LIN {X 0,Y 145.959,Z 433.252,A -85,B 0,C 180,E1 -25512.385,E2 -25512.385} C_VEL
LIN {X 0,Y 151.822,Z 425.901,A -85,B 0,C 180,E1 -25515.592,E2 -25515.592} C_VEL
LIN {X 0,Y 158.562,Z 416.452,A -85,B 0,C 180,E1 -25518.895,E2 -25518.895} C_VEL
LIN {X 0,Y 165.615,Z 405.723,A -85,B 0,C 180,E1 -25521.727,E2 -25521.727} C_VEL
LIN {X 0,Y 172.327,Z 394.008,A -85,B 0,C 180,E1 -25524.151,E2 -25524.151} C_VEL
LIN {X 0,Y 178.873,Z 380.825,A -85,B 0,C 180,E1 -25526.236,E2 -25526.236} C_VEL
LIN {X 0,Y 184.461,Z 367.074,A -85,B 0,C 180,E1 -25527.966,E2 -25527.966} C_VEL
LIN {X 0,Y 189.113,Z 353.283,A -85,B 0,C 180,E1 -25529.249,E2 -25529.249} C_VEL
LIN {X 0,Y 193.148,Z 337.834,A -85,B 0,C 180,E1 -25530.312,E2 -25530.312} C_VEL
LIN {X 0,Y 196.132,Z 321.975,A -85,B 0,C 180,E1 -25531.033,E2 -25531.033} C_VEL
LIN {X 0,Y 198.364,Z 301.16,A -85,B 0,C 180,E1 -25531.651,E2 -25531.651} C_VEL
LIN {X 0,Y 201.461,Z 266.459,A -85,B 0,C 180,E1 -25532.587,E2 -25532.587} C_VEL
LIN {X 0,Y 197.2,Z 257.514,A -85,B 0,C 180,E1 -25535.874,E2 -25535.874} C_VEL
LIN {X 0,Y 193.615,Z 250.815,A -85,B 0,C 180,E1 -25539.064,E2 -25539.064} C_VEL
LIN {X 0,Y 191.118,Z 246.438,A -85,B 0,C 180,E1 -25541.647,E2 -25541.647} C_VEL
LIN {X 0,Y 189.084,Z 243.025,A -85,B 0,C 180,E1 -25544.09,E2 -25544.09} C_VEL
LIN {X 0,Y 187.689,Z 240.639,A -85,B 0,C 180,E1 -25546.051,E2 -25546.051} C_VEL
LIN {X 0,Y 185.533,Z 236.807,A -85,B 0,C 180,E1 -25549.91,E2 -25549.91} C_VEL
LIN {X 0,Y 183.726,Z 233.495,A -85,B 0,C 180,E1 -25555.359,E2 -25555.359} C_VEL
LIN {X 0,Y 183.496,Z 232.327,A -85,B 0,C 180,E1 -25557.256,E2 -25557.256} C_VEL
LIN {X 0,Y 183.478,Z 232.249,A -85,B 0,C 180,E1 -25562.195,E2 -25562.195} C_VEL
LIN {X 0,Y 183.641,Z 233.069,A -85,B 0,C 180,E1 -25563.703,E2 -25563.703} C_VEL
LIN {X 0,Y 185.447,Z 236.708,A -85,B 0,C 180,E1 -25569.566,E2 -25569.566} C_VEL
LIN {X 0,Y 186.036,Z 237.651,A -85,B 0,C 180,E1 -25570.761,E2 -25570.761} C_VEL
LIN {X 0,Y 188.522,Z 241.906,A -85,B 0,C 180,E1 -25574.781,E2 -25574.781} C_VEL
LIN {X 0,Y 190.791,Z 245.771,A -85,B 0,C 180,E1 -25577.622,E2 -25577.622} C_VEL
LIN {X 0,Y 194.145,Z 251.69,A -85,B 0,C 180,E1 -25581.084,E2 -25581.084} C_VEL
LIN {X 0,Y 196.253,Z 256.423,A -85,B 0,C 180,E1 -25583.047,E2 -25583.047} C_VEL
LIN {X 0,Y 199.614,Z 265.237,A -85,B 0,C 180,E1 -25585.917,E2 -25585.917} C_VEL
LIN {X 0,Y 201.239,Z 269.895,A -85,B 0,C 180,E1 -25587.203,E2 -25587.203} C_VEL
LIN {X 0,Y 196.188,Z 324.073,A -85,B 0,C 180,E1 -25588.669,E2 -25588.669} C_VEL
LIN {X 0,Y 193.418,Z 339.856,A -85,B 0,C 180,E1 -25589.301,E2 -25589.301} C_VEL
LIN {X 0,Y 189.561,Z 355.077,A -85,B 0,C 180,E1 -25590.195,E2 -25590.195} C_VEL
LIN {X 0,Y 185.028,Z 368.798,A -85,B 0,C 180,E1 -25591.281,E2 -25591.281} C_VEL
LIN {X 0,Y 179.611,Z 382.244,A -85,B 0,C 180,E1 -25592.725,E2 -25592.725} C_VEL
LIN {X 0,Y 173.675,Z 394.769,A -85,B 0,C 180,E1 -25594.508,E2 -25594.508} C_VEL
LIN {X 0,Y 166.779,Z 407.28,A -85,B 0,C 180,E1 -25596.807,E2 -25596.807} C_VEL
LIN {X 0,Y 159.476,Z 418.758,A -85,B 0,C 180,E1 -25599.537,E2 -25599.537} C_VEL
LIN {X 0,Y 152.629,Z 428.424,A -85,B 0,C 180,E1 -25602.545,E2 -25602.545} C_VEL
LIN {X 0,Y 146.12,Z 436.937,A -85,B 0,C 180,E1 -25605.972,E2 -25605.972} C_VEL
LIN {X 0,Y 139.136,Z 445.526,A -85,B 0,C 180,E1 -25610.542,E2 -25610.542} C_VEL
LIN {X 0,Y 132.201,Z 453.257,A -85,B 0,C 180,E1 -25616.069,E2 -25616.069} C_VEL
LIN {X 0,Y 127.36,Z 458.667,A -85,B 0,C 180,E1 -25621.39,E2 -25621.39} C_VEL
LIN {X 0,Y 125.001,Z 460.669,A -85,B 0,C 180,E1 -25623.685,E2 -25623.685} C_VEL
LIN {X 0,Y 119.759,Z 463.482,A -85,B 0,C 180,E1 -25627.41,E2 -25627.41} C_VEL
LIN {X 0,Y 115.772,Z 465.343,A -85,B 0,C 180,E1 -25630.644,E2 -25630.644} C_VEL
LIN {X 0,Y 113.77,Z 466.536,A -85,B 0,C 180,E1 -25633.365,E2 -25633.365} C_VEL
LIN {X 0,Y 113.419,Z 466.836,A -85,B 0,C 180,E1 -25634.326,E2 -25634.326} C_VEL
LIN {X 0,Y 112.458,Z 468.336,A -85,B 0,C 180,E1 -25639.194,E2 -25639.194} C_VEL
LIN {X 0,Y 112.095,Z 469.523,A -85,B 0,C 180,E1 -25646.405,E2 -25646.405} C_VEL
LIN {X 0,Y 112.248,Z 469.683,A -85,B 0,C 180,E1 -25650,E2 -25650} C_VEL
LIN {X 0,Y 112.127,Z 469.052,A -85,B 0,C 180,E1 -25657.201,E2 -25657.201} C_VEL
LIN {X 0,Y 113.102,Z 467.265,A -85,B 0,C 180,E1 -25664.392,E2 -25664.392} C_VEL
LIN {X 0,Y 115.542,Z 464.307,A -85,B 0,C 180,E1 -25671.405,E2 -25671.405} C_VEL
LIN {X 0,Y 119.379,Z 460.108,A -85,B 0,C 180,E1 -25678.097,E2 -25678.097} C_VEL
LIN {X 0,Y 124.74,Z 454.565,A -85,B 0,C 180,E1 -25684.292,E2 -25684.292} C_VEL
LIN {X 0,Y 131.461,Z 447.53,A -85,B 0,C 180,E1 -25689.906,E2 -25689.906} C_VEL
LIN {X 0,Y 138.147,Z 439.961,A -85,B 0,C 180,E1 -25694.428,E2 -25694.428} C_VEL
LIN {X 0,Y 145.577,Z 430.948,A -85,B 0,C 180,E1 -25698.443,E2 -25698.443} C_VEL
LIN {X 0,Y 153.784,Z 420.066,A -85,B 0,C 180,E1 -25702.03,E2 -25702.03} C_VEL
LIN {X 0,Y 161.304,Z 408.87,A -85,B 0,C 180,E1 -25704.78,E2 -25704.78} C_VEL
LIN {X 0,Y 168.57,Z 396.421,A -85,B 0,C 180,E1 -25707.123,E2 -25707.123} C_VEL
LIN {X 0,Y 175.185,Z 383.102,A -85,B 0,C 180,E1 -25709.039,E2 -25709.039} C_VEL
LIN {X 0,Y 180.735,Z 369.84,A -85,B 0,C 180,E1 -25710.467,E2 -25710.467} C_VEL
LIN {X 0,Y 185.714,Z 355.323,A -85,B 0,C 180,E1 -25711.625,E2 -25711.625} C_VEL
LIN {X 0,Y 189.658,Z 340.259,A -85,B 0,C 180,E1 -25712.503,E2 -25712.503} C_VEL
LIN {X 0,Y 192.438,Z 324.99,A -85,B 0,C 180,E1 -25713.123,E2 -25713.123} C_VEL
LIN {X 0,Y 196.109,Z 288.872,A -85,B 0,C 180,E1 -25714.062,E2 -25714.062} C_VEL
LIN {X 0,Y 197.581,Z 272.685,A -85,B 0,C 180,E1 -25714.504,E2 -25714.504} C_VEL
LIN {X 0,Y 194.287,Z 263.272,A -85,B 0,C 180,E1 -25717.468,E2 -25717.468} C_VEL
LIN {X 0,Y 192.199,Z 258.069,A -85,B 0,C 180,E1 -25719.533,E2 -25719.533} C_VEL
LIN {X 0,Y 189.081,Z 252.283,A -85,B 0,C 180,E1 -25722.91,E2 -25722.91} C_VEL
LIN {X 0,Y 186.331,Z 247.346,A -85,B 0,C 180,E1 -25726.643,E2 -25726.643} C_VEL
LIN {X 0,Y 184.285,Z 243.616,A -85,B 0,C 180,E1 -25730.396,E2 -25730.396} C_VEL
LIN {X 0,Y 182.602,Z 240.468,A -85,B 0,C 180,E1 -25735.447,E2 -25735.447} C_VEL
LIN {X 0,Y 182.361,Z 239.282,A -85,B 0,C 180,E1 -25737.239,E2 -25737.239} C_VEL
LIN {X 0,Y 182.233,Z 239.216,A -85,B 0,C 180,E1 -25742.21,E2 -25742.21} C_VEL
LIN {X 0,Y 182.442,Z 239.623,A -85,B 0,C 180,E1 -25743.866,E2 -25743.866} C_VEL
LIN {X 0,Y 183.716,Z 242.998,A -85,B 0,C 180,E1 -25748.802,E2 -25748.802} C_VEL
LIN {X 0,Y 184.522,Z 244.089,A -85,B 0,C 180,E1 -25750.562,E2 -25750.562} C_VEL
LIN {X 0,Y 186.922,Z 248.505,A -85,B 0,C 180,E1 -25754.702,E2 -25754.702} C_VEL
LIN {X 0,Y 189.301,Z 252.766,A -85,B 0,C 180,E1 -25757.8,E2 -25757.8} C_VEL
LIN {X 0,Y 192.242,Z 258.192,A -85,B 0,C 180,E1 -25760.952,E2 -25760.952} C_VEL
LIN {X 0,Y 195.843,Z 265.523,A -85,B 0,C 180,E1 -25764.233,E2 -25764.233} C_VEL
LIN {X 0,Y 197.761,Z 269.785,A -85,B 0,C 180,E1 -25765.805,E2 -25765.805} C_VEL
LIN {X 0,Y 192.923,Z 319.693,A -85,B 0,C 180,E1 -25767.155,E2 -25767.155} C_VEL
LIN {X 0,Y 190.163,Z 335.085,A -85,B 0,C 180,E1 -25767.788,E2 -25767.788} C_VEL
LIN {X 0,Y 186.696,Z 349.013,A -85,B 0,C 180,E1 -25768.648,E2 -25768.648} C_VEL
LIN {X 0,Y 182.267,Z 362.803,A -85,B 0,C 180,E1 -25769.822,E2 -25769.822} C_VEL
LIN {X 0,Y 176.796,Z 376.715,A -85,B 0,C 180,E1 -25771.409,E2 -25771.409} C_VEL
LIN {X 0,Y 170.343,Z 390.076,A -85,B 0,C 180,E1 -25773.335,E2 -25773.335} C_VEL
LIN {X 0,Y 163.244,Z 402.48,A -85,B 0,C 180,E1 -25775.648,E2 -25775.648} C_VEL
LIN {X 0,Y 156.47,Z 412.863,A -85,B 0,C 180,E1 -25778.184,E2 -25778.184} C_VEL
LIN {X 0,Y 149.056,Z 422.901,A -85,B 0,C 180,E1 -25781.308,E2 -25781.308} C_VEL
LIN {X 0,Y 143.024,Z 430.701,A -85,B 0,C 180,E1 -25784.56,E2 -25784.56} C_VEL
LIN {X 0,Y 135.901,Z 438.777,A -85,B 0,C 180,E1 -25788.749,E2 -25788.749} C_VEL
LIN {X 0,Y 129.575,Z 445.438,A -85,B 0,C 180,E1 -25793.371,E2 -25793.371} C_VEL
LIN {X 0,Y 123.479,Z 451.594,A -85,B 0,C 180,E1 -25799.186,E2 -25799.186} C_VEL
LIN {X 0,Y 118.72,Z 456.337,A -85,B 0,C 180,E1 -25805.519,E2 -25805.519} C_VEL
LIN {X 0,Y 115.274,Z 459.803,A -85,B 0,C 180,E1 -25812.252,E2 -25812.252} C_VEL
LIN {X 0,Y 113.203,Z 462.086,A -85,B 0,C 180,E1 -25819.266,E2 -25819.266} C_VEL
LIN {X 0,Y 112.353,Z 463.242,A -85,B 0,C 180,E1 -25826.414,E2 -25826.414} C_VEL
LIN {X 0,Y 112.335,Z 463.394,A -85,B 0,C 180,E1 -25830,E2 -25830} C_VEL
LIN {X 0,Y 112.624,Z 462.835,A -85,B 0,C 180,E1 -25837.17,E2 -25837.17} C_VEL
LIN {X 0,Y 114.052,Z 461.162,A -85,B 0,C 180,E1 -25844.27,E2 -25844.27} C_VEL
LIN {X 0,Y 116.719,Z 458.337,A -85,B 0,C 180,E1 -25851.179,E2 -25851.179} C_VEL
LIN {X 0,Y 120.935,Z 454.278,A -85,B 0,C 180,E1 -25857.705,E2 -25857.705} C_VEL
LIN {X 0,Y 126.325,Z 448.897,A -85,B 0,C 180,E1 -25863.804,E2 -25863.804} C_VEL
LIN {X 0,Y 133.008,Z 442.029,A -85,B 0,C 180,E1 -25869.351,E2 -25869.351} C_VEL
LIN {X 0,Y 140.793,Z 433.449,A -85,B 0,C 180,E1 -25874.335,E2 -25874.335} C_VEL
LIN {X 0,Y 148.072,Z 424.61,A -85,B 0,C 180,E1 -25878.181,E2 -25878.181} C_VEL
LIN {X 0,Y 155.16,Z 415.03,A -85,B 0,C 180,E1 -25881.384,E2 -25881.384} C_VEL
LIN {X 0,Y 163.16,Z 402.982,A -85,B 0,C 180,E1 -25884.393,E2 -25884.393} C_VEL
LIN {X 0,Y 170.262,Z 390.675,A -85,B 0,C 180,E1 -25886.707,E2 -25886.707} C_VEL
LIN {X 0,Y 176.338,Z 378.186,A -85,B 0,C 180,E1 -25888.564,E2 -25888.564} C_VEL
LIN {X 0,Y 181.489,Z 365.505,A -85,B 0,C 180,E1 -25890.049,E2 -25890.049} C_VEL
LIN {X 0,Y 185.95,Z 352.346,A -85,B 0,C 180,E1 -25891.209,E2 -25891.209} C_VEL
LIN {X 0,Y 189.92,Z 337.261,A -85,B 0,C 180,E1 -25892.21,E2 -25892.21} C_VEL
LIN {X 0,Y 192.89,Z 321.585,A -85,B 0,C 180,E1 -25892.896,E2 -25892.896} C_VEL
LIN {X 0,Y 195.23,Z 299.87,A -85,B 0,C 180,E1 -25893.524,E2 -25893.524} C_VEL
LIN {X 0,Y 198.036,Z 270.016,A -85,B 0,C 180,E1 -25894.286,E2 -25894.286} C_VEL
LIN {X 0,Y 194.311,Z 262.063,A -85,B 0,C 180,E1 -25897.435,E2 -25897.435} C_VEL
LIN {X 0,Y 191.087,Z 255.8,A -85,B 0,C 180,E1 -25900.6,E2 -25900.6} C_VEL
LIN {X 0,Y 188.294,Z 250.735,A -85,B 0,C 180,E1 -25903.883,E2 -25903.883} C_VEL
LIN {X 0,Y 186.382,Z 247.347,A -85,B 0,C 180,E1 -25906.639,E2 -25906.639} C_VEL
LIN {X 0,Y 184.409,Z 243.664,A -85,B 0,C 180,E1 -25910.402,E2 -25910.402} C_VEL
LIN {X 0,Y 182.727,Z 240.167,A -85,B 0,C 180,E1 -25916.14,E2 -25916.14} C_VEL
LIN {X 0,Y 182.572,Z 239.291,A -85,B 0,C 180,E1 -25917.794,E2 -25917.794} C_VEL
LIN {X 0,Y 182.613,Z 239.299,A -85,B 0,C 180,E1 -25922.205,E2 -25922.205} C_VEL
LIN {X 0,Y 184.443,Z 243.691,A -85,B 0,C 180,E1 -25929.319,E2 -25929.319} C_VEL
LIN {X 0,Y 187.034,Z 248.381,A -85,B 0,C 180,E1 -25933.998,E2 -25933.998} C_VEL
LIN {X 0,Y 189.551,Z 252.95,A -85,B 0,C 180,E1 -25937.324,E2 -25937.324} C_VEL
LIN {X 0,Y 192.628,Z 258.726,A -85,B 0,C 180,E1 -25940.628,E2 -25940.628} C_VEL
LIN {X 0,Y 195.09,Z 265.052,A -85,B 0,C 180,E1 -25943.041,E2 -25943.041} C_VEL
LIN {X 0,Y 197.804,Z 272.967,A -85,B 0,C 180,E1 -25945.468,E2 -25945.468} C_VEL
LIN {X 0,Y 192.857,Z 324.071,A -85,B 0,C 180,E1 -25946.826,E2 -25946.826} C_VEL
LIN {X 0,Y 190.168,Z 339.2,A -85,B 0,C 180,E1 -25947.419,E2 -25947.419} C_VEL
LIN {X 0,Y 186.09,Z 354.885,A -85,B 0,C 180,E1 -25948.304,E2 -25948.304} C_VEL
LIN {X 0,Y 181.444,Z 368.605,A -85,B 0,C 180,E1 -25949.365,E2 -25949.365} C_VEL
LIN {X 0,Y 175.871,Z 382.05,A -85,B 0,C 180,E1 -25950.777,E2 -25950.777} C_VEL
LIN {X 0,Y 169.333,Z 395.376,A -85,B 0,C 180,E1 -25952.653,E2 -25952.653} C_VEL
LIN {X 0,Y 161.965,Z 408.156,A -85,B 0,C 180,E1 -25955.012,E2 -25955.012} C_VEL
LIN {X 0,Y 153.81,Z 420.321,A -85,B 0,C 180,E1 -25957.982,E2 -25957.982} C_VEL
LIN {X 0,Y 145.602,Z 431.152,A -85,B 0,C 180,E1 -25961.568,E2 -25961.568} C_VEL
LIN {X 0,Y 138.413,Z 439.903,A -85,B 0,C 180,E1 -25965.472,E2 -25965.472} C_VEL
LIN {X 0,Y 131.53,Z 447.689,A -85,B 0,C 180,E1 -25970.119,E2 -25970.119} C_VEL
LIN {X 0,Y 126.304,Z 453.057,A -85,B 0,C 180,E1 -25974.249,E2 -25974.249} C_VEL
LIN {X 0,Y 120.674,Z 458.941,A -85,B 0,C 180,E1 -25980.328,E2 -25980.328} C_VEL
LIN {X 0,Y 117.361,Z 462.447,A -85,B 0,C 180,E1 -25985.217,E2 -25985.217} C_VEL
LIN {X 0,Y 114.102,Z 465.992,A -85,B 0,C 180,E1 -25992.063,E2 -25992.063} C_VEL
LIN {X 0,Y 113.419,Z 466.836,A -85,B 0,C 180,E1 -25994.326,E2 -25994.326} C_VEL
LIN {X 0,Y 112.197,Z 467.831,A -85,B 0,C 180,E1 -25997.215,E2 -25997.215} C_VEL
LIN {X 0,Y 108.996,Z 468.969,A -85,B 0,C 180,E1 -26002.024,E2 -26002.024} C_VEL
LIN {X 0,Y 105.595,Z 469.508,A -85,B 0,C 180,E1 -26008.165,E2 -26008.165} C_VEL
LIN {X 0,Y 105.134,Z 469.471,A -85,B 0,C 180,E1 -26010.321,E2 -26010.321} C_VEL
LIN {X 0,Y 105.053,Z 468.852,A -85,B 0,C 180,E1 -26017.689,E2 -26017.689} C_VEL
LIN {X 0,Y 106.184,Z 467.064,A -85,B 0,C 180,E1 -26025.352,E2 -26025.352} C_VEL
LIN {X 0,Y 108.884,Z 464.105,A -85,B 0,C 180,E1 -26032.785,E2 -26032.785} C_VEL
LIN {X 0,Y 113.108,Z 459.907,A -85,B 0,C 180,E1 -26039.807,E2 -26039.807} C_VEL
LIN {X 0,Y 118.877,Z 454.363,A -85,B 0,C 180,E1 -26046.242,E2 -26046.242} C_VEL
LIN {X 0,Y 126.045,Z 447.327,A -85,B 0,C 180,E1 -26051.997,E2 -26051.997} C_VEL
LIN {X 0,Y 133.556,Z 439.265,A -85,B 0,C 180,E1 -26056.836,E2 -26056.836} C_VEL
LIN {X 0,Y 140.943,Z 430.746,A -85,B 0,C 180,E1 -26060.615,E2 -26060.615} C_VEL
LIN {X 0,Y 149.492,Z 419.863,A -85,B 0,C 180,E1 -26064.191,E2 -26064.191} C_VEL
LIN {X 0,Y 157.306,Z 408.668,A -85,B 0,C 180,E1 -26066.898,E2 -26066.898} C_VEL
LIN {X 0,Y 165.108,Z 395.702,A -85,B 0,C 180,E1 -26069.284,E2 -26069.284} C_VEL
LIN {X 0,Y 171.627,Z 382.898,A -85,B 0,C 180,E1 -26071.08,E2 -26071.08} C_VEL
LIN {X 0,Y 177.332,Z 369.635,A -85,B 0,C 180,E1 -26072.469,E2 -26072.469} C_VEL
LIN {X 0,Y 182.448,Z 355.117,A -85,B 0,C 180,E1 -26073.586,E2 -26073.586} C_VEL
LIN {X 0,Y 186.488,Z 340.051,A -85,B 0,C 180,E1 -26074.437,E2 -26074.437} C_VEL
LIN {X 0,Y 189.259,Z 325.22,A -85,B 0,C 180,E1 -26075.028,E2 -26075.028} C_VEL
LIN {X 0,Y 192.307,Z 296.736,A -85,B 0,C 180,E1 -26075.769,E2 -26075.769} C_VEL
LIN {X 0,Y 194.306,Z 275.86,A -85,B 0,C 180,E1 -26076.304,E2 -26076.304} C_VEL
LIN {X 0,Y 191.694,Z 267.952,A -85,B 0,C 180,E1 -26078.915,E2 -26078.915} C_VEL
LIN {X 0,Y 190.099,Z 263.817,A -85,B 0,C 180,E1 -26080.636,E2 -26080.636} C_VEL
LIN {X 0,Y 186.9,Z 257.529,A -85,B 0,C 180,E1 -26084.46,E2 -26084.46} C_VEL
LIN {X 0,Y 184.856,Z 253.826,A -85,B 0,C 180,E1 -26087.512,E2 -26087.512} C_VEL
LIN {X 0,Y 183.132,Z 250.42,A -85,B 0,C 180,E1 -26090.961,E2 -26090.961} C_VEL
LIN {X 0,Y 181.628,Z 247.298,A -85,B 0,C 180,E1 -26095.979,E2 -26095.979} C_VEL
LIN {X 0,Y 181.494,Z 246.355,A -85,B 0,C 180,E1 -26097.226,E2 -26097.226} C_VEL
LIN {X 0,Y 181.279,Z 246.096,A -85,B 0,C 180,E1 -26100,E2 -26100} C_VEL
LIN {X 0,Y 181.526,Z 246.656,A -85,B 0,C 180,E1 -26103.607,E2 -26103.607} C_VEL
LIN {X 0,Y 182.764,Z 250.033,A -85,B 0,C 180,E1 -26108.639,E2 -26108.639} C_VEL
LIN {X 0,Y 183.445,Z 251.083,A -85,B 0,C 180,E1 -26110.206,E2 -26110.206} C_VEL
LIN {X 0,Y 185.533,Z 255.12,A -85,B 0,C 180,E1 -26114.029,E2 -26114.029} C_VEL
LIN {X 0,Y 187.886,Z 259.548,A -85,B 0,C 180,E1 -26117.272,E2 -26117.272} C_VEL
LIN {X 0,Y 190.91,Z 265.585,A -85,B 0,C 180,E1 -26120.664,E2 -26120.664} C_VEL
LIN {X 0,Y 193.676,Z 271.568,A -85,B 0,C 180,E1 -26123.317,E2 -26123.317} C_VEL
LIN {X 0,Y 194.461,Z 273.393,A -85,B 0,C 180,E1 -26124.018,E2 -26124.018} C_VEL
LIN {X 0,Y 189.888,Z 319.327,A -85,B 0,C 180,E1 -26125.232,E2 -26125.232} C_VEL
LIN {X 0,Y 187.153,Z 334.525,A -85,B 0,C 180,E1 -26125.831,E2 -26125.831} C_VEL
LIN {X 0,Y 183.411,Z 349.218,A -85,B 0,C 180,E1 -26126.709,E2 -26126.709} C_VEL
LIN {X 0,Y 178.839,Z 363.009,A -85,B 0,C 180,E1 -26127.846,E2 -26127.846} C_VEL
LIN {X 0,Y 173.371,Z 376.476,A -85,B 0,C 180,E1 -26129.337,E2 -26129.337} C_VEL
LIN {X 0,Y 167.212,Z 388.993,A -85,B 0,C 180,E1 -26131.088,E2 -26131.088} C_VEL
LIN {X 0,Y 159.84,Z 401.62,A -85,B 0,C 180,E1 -26133.341,E2 -26133.341} C_VEL
LIN {X 0,Y 152.187,Z 413.065,A -85,B 0,C 180,E1 -26136.084,E2 -26136.084} C_VEL
LIN {X 0,Y 144.08,Z 423.573,A -85,B 0,C 180,E1 -26139.355,E2 -26139.355} C_VEL
LIN {X 0,Y 136.996,Z 432.126,A -85,B 0,C 180,E1 -26143.027,E2 -26143.027} C_VEL
LIN {X 0,Y 129.619,Z 439.979,A -85,B 0,C 180,E1 -26147.331,E2 -26147.331} C_VEL
LIN {X 0,Y 122.176,Z 447.304,A -85,B 0,C 180,E1 -26152.843,E2 -26152.843} C_VEL
LIN {X 0,Y 115.98,Z 453.107,A -85,B 0,C 180,E1 -26158.998,E2 -26158.998} C_VEL
LIN {X 0,Y 112.283,Z 456.537,A -85,B 0,C 180,E1 -26164.015,E2 -26164.015} C_VEL
LIN {X 0,Y 108.496,Z 460.004,A -85,B 0,C 180,E1 -26171.102,E2 -26171.102} C_VEL
LIN {X 0,Y 106.216,Z 462.286,A -85,B 0,C 180,E1 -26178.551,E2 -26178.551} C_VEL
LIN {X 0,Y 105.265,Z 463.441,A -85,B 0,C 180,E1 -26186.172,E2 -26186.172} C_VEL
LIN {X 0,Y 105.237,Z 463.593,A -85,B 0,C 180,E1 -26190,E2 -26190} C_VEL
LIN {X 0,Y 105.593,Z 463.033,A -85,B 0,C 180,E1 -26197.65,E2 -26197.65} C_VEL
LIN {X 0,Y 107.158,Z 461.361,A -85,B 0,C 180,E1 -26205.209,E2 -26205.209} C_VEL
LIN {X 0,Y 110.095,Z 458.536,A -85,B 0,C 180,E1 -26212.521,E2 -26212.521} C_VEL
LIN {X 0,Y 114.638,Z 454.478,A -85,B 0,C 180,E1 -26219.37,E2 -26219.37} C_VEL
LIN {X 0,Y 120.451,Z 449.095,A -85,B 0,C 180,E1 -26225.696,E2 -26225.696} C_VEL
LIN {X 0,Y 127.581,Z 442.227,A -85,B 0,C 180,E1 -26231.38,E2 -26231.38} C_VEL
LIN {X 0,Y 134.691,Z 434.842,A -85,B 0,C 180,E1 -26235.845,E2 -26235.845} C_VEL
LIN {X 0,Y 141.637,Z 426.963,A -85,B 0,C 180,E1 -26239.429,E2 -26239.429} C_VEL
LIN {X 0,Y 148.348,Z 418.465,A -85,B 0,C 180,E1 -26242.517,E2 -26242.517} C_VEL
LIN {X 0,Y 155.929,Z 408.058,A -85,B 0,C 180,E1 -26245.343,E2 -26245.343} C_VEL
LIN {X 0,Y 163.074,Z 396.737,A -85,B 0,C 180,E1 -26247.756,E2 -26247.756} C_VEL
LIN {X 0,Y 169.839,Z 384.428,A -85,B 0,C 180,E1 -26249.748,E2 -26249.748} C_VEL
LIN {X 0,Y 175.972,Z 370.965,A -85,B 0,C 180,E1 -26251.48,E2 -26251.48} C_VEL
LIN {X 0,Y 181.206,Z 357,A -85,B 0,C 180,E1 -26252.826,E2 -26252.826} C_VEL
LIN {X 0,Y 185.49,Z 342.639,A -85,B 0,C 180,E1 -26253.831,E2 -26253.831} C_VEL
LIN {X 0,Y 188.76,Z 327.829,A -85,B 0,C 180,E1 -26254.576,E2 -26254.576} C_VEL
LIN {X 0,Y 191.009,Z 312.004,A -85,B 0,C 180,E1 -26255.111,E2 -26255.111} C_VEL
LIN {X 0,Y 194.707,Z 273.571,A -85,B 0,C 180,E1 -26256.098,E2 -26256.098} C_VEL
LIN {X 0,Y 191.419,Z 266.286,A -85,B 0,C 180,E1 -26259.194,E2 -26259.194} C_VEL
LIN {X 0,Y 188.424,Z 260.334,A -85,B 0,C 180,E1 -26262.499,E2 -26262.499} C_VEL
LIN {X 0,Y 186.354,Z 256.478,A -85,B 0,C 180,E1 -26265.238,E2 -26265.238} C_VEL
LIN {X 0,Y 185.084,Z 254.064,A -85,B 0,C 180,E1 -26267.249,E2 -26267.249} C_VEL
LIN {X 0,Y 183.296,Z 250.539,A -85,B 0,C 180,E1 -26270.899,E2 -26270.899} C_VEL
LIN {X 0,Y 181.769,Z 246.756,A -85,B 0,C 180,E1 -26276.952,E2 -26276.952} C_VEL
LIN {X 0,Y 181.705,Z 246.353,A -85,B 0,C 180,E1 -26277.783,E2 -26277.783} C_VEL
LIN {X 0,Y 181.743,Z 246.395,A -85,B 0,C 180,E1 -26282.216,E2 -26282.216} C_VEL
LIN {X 0,Y 183.21,Z 250.417,A -85,B 0,C 180,E1 -26288.548,E2 -26288.548} C_VEL
LIN {X 0,Y 183.796,Z 251.506,A -85,B 0,C 180,E1 -26289.908,E2 -26289.908} C_VEL
LIN {X 0,Y 185.704,Z 255.116,A -85,B 0,C 180,E1 -26293.403,E2 -26293.403} C_VEL
LIN {X 0,Y 188.056,Z 259.604,A -85,B 0,C 180,E1 -26296.696,E2 -26296.696} C_VEL
LIN {X 0,Y 190.88,Z 265.244,A -85,B 0,C 180,E1 -26299.912,E2 -26299.912} C_VEL
LIN {X 0,Y 193.413,Z 272.592,A -85,B 0,C 180,E1 -26302.574,E2 -26302.574} C_VEL
LIN {X 0,Y 194.527,Z 276.013,A -85,B 0,C 180,E1 -26303.652,E2 -26303.652} C_VEL
LIN {X 0,Y 189.733,Z 324.051,A -85,B 0,C 180,E1 -26304.919,E2 -26304.919} C_VEL
LIN {X 0,Y 186.885,Z 339.478,A -85,B 0,C 180,E1 -26305.505,E2 -26305.505} C_VEL
LIN {X 0,Y 182.829,Z 354.693,A -85,B 0,C 180,E1 -26306.344,E2 -26306.344} C_VEL
LIN {X 0,Y 178.071,Z 368.412,A -85,B 0,C 180,E1 -26307.374,E2 -26307.374} C_VEL
LIN {X 0,Y 172.329,Z 381.855,A -85,B 0,C 180,E1 -26308.738,E2 -26308.738} C_VEL
LIN {X 0,Y 165.924,Z 394.555,A -85,B 0,C 180,E1 -26310.479,E2 -26310.479} C_VEL
LIN {X 0,Y 158.651,Z 406.888,A -85,B 0,C 180,E1 -26312.683,E2 -26312.683} C_VEL
LIN {X 0,Y 150.778,Z 418.363,A -85,B 0,C 180,E1 -26315.343,E2 -26315.343} C_VEL
LIN {X 0,Y 143.339,Z 428.028,A -85,B 0,C 180,E1 -26318.326,E2 -26318.326} C_VEL
LIN {X 0,Y 135.276,Z 437.531,A -85,B 0,C 180,E1 -26322.24,E2 -26322.24} C_VEL
LIN {X 0,Y 128.065,Z 445.458,A -85,B 0,C 180,E1 -26326.687,E2 -26326.687} C_VEL
LIN {X 0,Y 120.559,Z 452.858,A -85,B 0,C 180,E1 -26332.258,E2 -26332.258} C_VEL
LIN {X 0,Y 114.487,Z 458.741,A -85,B 0,C 180,E1 -26338.547,E2 -26338.547} C_VEL
LIN {X 0,Y 110.903,Z 462.248,A -85,B 0,C 180,E1 -26343.666,E2 -26343.666} C_VEL
LIN {X 0,Y 107.319,Z 465.792,A -85,B 0,C 180,E1 -26350.887,E2 -26350.887} C_VEL
LIN {X 0,Y 105.463,Z 468.137,A -85,B 0,C 180,E1 -26358.468,E2 -26358.468} C_VEL
LIN {X 0,Y 105.005,Z 469.324,A -85,B 0,C 180,E1 -26366.162,E2 -26366.162} C_VEL
LIN {X 0,Y 105.134,Z 469.471,A -85,B 0,C 180,E1 -26370.321,E2 -26370.321} C_VEL
LIN {X 0,Y 104.271,Z 469.314,A -85,B 0,C 180,E1 -26373.515,E2 -26373.515} C_VEL
LIN {X 0,Y 101.541,Z 468.64,A -85,B 0,C 180,E1 -26378.815,E2 -26378.815} C_VEL
LIN {X 0,Y 99.692,Z 467.731,A -85,B 0,C 180,E1 -26383.222,E2 -26383.222} C_VEL
LIN {X 0,Y 99.406,Z 466.816,A -85,B 0,C 180,E1 -26386.608,E2 -26386.608} C_VEL
LIN {X 0,Y 99.638,Z 466.442,A -85,B 0,C 180,E1 -26387.725,E2 -26387.725} C_VEL
LIN {X 0,Y 102.3,Z 463.903,A -85,B 0,C 180,E1 -26394.343,E2 -26394.343} C_VEL
LIN {X 0,Y 106.942,Z 459.705,A -85,B 0,C 180,E1 -26401.718,E2 -26401.718} C_VEL
LIN {X 0,Y 113.158,Z 454.161,A -85,B 0,C 180,E1 -26408.395,E2 -26408.395} C_VEL
LIN {X 0,Y 120.825,Z 447.126,A -85,B 0,C 180,E1 -26414.267,E2 -26414.267} C_VEL
LIN {X 0,Y 128.169,Z 439.682,A -85,B 0,C 180,E1 -26418.852,E2 -26418.852} C_VEL
LIN {X 0,Y 136.511,Z 430.543,A -85,B 0,C 180,E1 -26422.938,E2 -26422.938} C_VEL
LIN {X 0,Y 145.416,Z 419.66,A -85,B 0,C 180,E1 -26426.481,E2 -26426.481} C_VEL
LIN {X 0,Y 154.229,Z 407.43,A -85,B 0,C 180,E1 -26429.329,E2 -26429.329} C_VEL
LIN {X 0,Y 161.719,Z 395.216,A -85,B 0,C 180,E1 -26431.514,E2 -26431.514} C_VEL
LIN {X 0,Y 168.298,Z 382.694,A -85,B 0,C 180,E1 -26433.203,E2 -26433.203} C_VEL
LIN {X 0,Y 174.157,Z 369.43,A -85,B 0,C 180,E1 -26434.546,E2 -26434.546} C_VEL
LIN {X 0,Y 179.395,Z 354.911,A -85,B 0,C 180,E1 -26435.622,E2 -26435.622} C_VEL
LIN {X 0,Y 183.54,Z 339.843,A -85,B 0,C 180,E1 -26436.434,E2 -26436.434} C_VEL
LIN {X 0,Y 186.455,Z 324.525,A -85,B 0,C 180,E1 -26437.021,E2 -26437.021} C_VEL
LIN {X 0,Y 190.395,Z 287.773,A -85,B 0,C 180,E1 -26437.923,E2 -26437.923} C_VEL
LIN {X 0,Y 191.235,Z 279.063,A -85,B 0,C 180,E1 -26438.155,E2 -26438.155} C_VEL
LIN {X 0,Y 188.899,Z 271.64,A -85,B 0,C 180,E1 -26440.79,E2 -26440.79} C_VEL
LIN {X 0,Y 186.838,Z 266.97,A -85,B 0,C 180,E1 -26443.262,E2 -26443.262} C_VEL
LIN {X 0,Y 184.704,Z 262.733,A -85,B 0,C 180,E1 -26446.243,E2 -26446.243} C_VEL
LIN {X 0,Y 183.284,Z 260,A -85,B 0,C 180,E1 -26448.667,E2 -26448.667} C_VEL
LIN {X 0,Y 182.055,Z 257.306,A -85,B 0,C 180,E1 -26451.397,E2 -26451.397} C_VEL
LIN {X 0,Y 180.654,Z 254.028,A -85,B 0,C 180,E1 -26456.655,E2 -26456.655} C_VEL
LIN {X 0,Y 180.559,Z 253.298,A -85,B 0,C 180,E1 -26457.77,E2 -26457.77} C_VEL
LIN {X 0,Y 180.502,Z 253.322,A -85,B 0,C 180,E1 -26462.232,E2 -26462.232} C_VEL
LIN {X 0,Y 180.623,Z 253.821,A -85,B 0,C 180,E1 -26463.486,E2 -26463.486} C_VEL
LIN {X 0,Y 181.897,Z 257.182,A -85,B 0,C 180,E1 -26468.681,E2 -26468.681} C_VEL
LIN {X 0,Y 182.428,Z 258.249,A -85,B 0,C 180,E1 -26469.984,E2 -26469.984} C_VEL
LIN {X 0,Y 184.187,Z 261.777,A -85,B 0,C 180,E1 -26473.375,E2 -26473.375} C_VEL
LIN {X 0,Y 186.111,Z 265.61,A -85,B 0,C 180,E1 -26476.241,E2 -26476.241} C_VEL
LIN {X 0,Y 188.905,Z 271.487,A -85,B 0,C 180,E1 -26479.637,E2 -26479.637} C_VEL
LIN {X 0,Y 191.338,Z 277.056,A -85,B 0,C 180,E1 -26482.163,E2 -26482.163} C_VEL
LIN {X 0,Y 186.907,Z 319.966,A -85,B 0,C 180,E1 -26483.281,E2 -26483.281} C_VEL
LIN {X 0,Y 184.181,Z 334.733,A -85,B 0,C 180,E1 -26483.85,E2 -26483.85} C_VEL
LIN {X 0,Y 179.962,Z 350.576,A -85,B 0,C 180,E1 -26484.773,E2 -26484.773} C_VEL
LIN {X 0,Y 174.936,Z 365.069,A -85,B 0,C 180,E1 -26485.985,E2 -26485.985} C_VEL
LIN {X 0,Y 169.022,Z 378.845,A -85,B 0,C 180,E1 -26487.533,E2 -26487.533} C_VEL
LIN {X 0,Y 162.286,Z 391.719,A -85,B 0,C 180,E1 -26489.362,E2 -26489.362} C_VEL
LIN {X 0,Y 154.71,Z 403.92,A -85,B 0,C 180,E1 -26491.596,E2 -26491.596} C_VEL
LIN {X 0,Y 146.799,Z 415.032,A -85,B 0,C 180,E1 -26494.325,E2 -26494.325} C_VEL
LIN {X 0,Y 138.223,Z 425.571,A -85,B 0,C 180,E1 -26497.778,E2 -26497.778} C_VEL
LIN {X 0,Y 131.073,Z 433.55,A -85,B 0,C 180,E1 -26501.352,E2 -26501.352} C_VEL
LIN {X 0,Y 123.433,Z 441.18,A -85,B 0,C 180,E1 -26505.774,E2 -26505.774} C_VEL
LIN {X 0,Y 116.565,Z 447.506,A -85,B 0,C 180,E1 -26510.723,E2 -26510.723} C_VEL
LIN {X 0,Y 109.923,Z 453.308,A -85,B 0,C 180,E1 -26517.081,E2 -26517.081} C_VEL
LIN {X 0,Y 105.917,Z 456.737,A -85,B 0,C 180,E1 -26522.324,E2 -26522.324} C_VEL
LIN {X 0,Y 101.776,Z 460.204,A -85,B 0,C 180,E1 -26529.802,E2 -26529.802} C_VEL
LIN {X 0,Y 99.262,Z 462.485,A -85,B 0,C 180,E1 -26537.737,E2 -26537.737} C_VEL
LIN {X 0,Y 98.189,Z 463.64,A -85,B 0,C 180,E1 -26545.896,E2 -26545.896} C_VEL
LIN {X 0,Y 98.151,Z 463.791,A -85,B 0,C 180,E1 -26550,E2 -26550} C_VEL
LIN {X 0,Y 98.553,Z 463.232,A -85,B 0,C 180,E1 -26558.2,E2 -26558.2} C_VEL
LIN {X 0,Y 100.308,Z 461.56,A -85,B 0,C 180,E1 -26566.276,E2 -26566.276} C_VEL
LIN {X 0,Y 103.541,Z 458.735,A -85,B 0,C 180,E1 -26574.033,E2 -26574.033} C_VEL
LIN {X 0,Y 108.454,Z 454.678,A -85,B 0,C 180,E1 -26581.226,E2 -26581.226} C_VEL
LIN {X 0,Y 114.73,Z 449.294,A -85,B 0,C 180,E1 -26587.776,E2 -26587.776} C_VEL
LIN {X 0,Y 122.322,Z 442.424,A -85,B 0,C 180,E1 -26593.588,E2 -26593.588} C_VEL
LIN {X 0,Y 129.836,Z 435.039,A -85,B 0,C 180,E1 -26598.098,E2 -26598.098} C_VEL
LIN {X 0,Y 138.18,Z 425.917,A -85,B 0,C 180,E1 -26602.22,E2 -26602.22} C_VEL
LIN {X 0,Y 145.406,Z 417.042,A -85,B 0,C 180,E1 -26605.253,E2 -26605.253} C_VEL
LIN {X 0,Y 153.298,Z 406.312,A -85,B 0,C 180,E1 -26608.01,E2 -26608.01} C_VEL
LIN {X 0,Y 160.782,Z 394.593,A -85,B 0,C 180,E1 -26610.316,E2 -26610.316} C_VEL
LIN {X 0,Y 167.743,Z 381.869,A -85,B 0,C 180,E1 -26612.226,E2 -26612.226} C_VEL
LIN {X 0,Y 173.396,Z 369.414,A -85,B 0,C 180,E1 -26613.736,E2 -26613.736} C_VEL
LIN {X 0,Y 178.807,Z 354.984,A -85,B 0,C 180,E1 -26615.023,E2 -26615.023} C_VEL
LIN {X 0,Y 183.018,Z 340.681,A -85,B 0,C 180,E1 -26615.955,E2 -26615.955} C_VEL
LIN {X 0,Y 186.31,Z 325.296,A -85,B 0,C 180,E1 -26616.658,E2 -26616.658} C_VEL
LIN {X 0,Y 188.36,Z 310.076,A -85,B 0,C 180,E1 -26617.123,E2 -26617.123} C_VEL
LIN {X 0,Y 191.592,Z 277.341,A -85,B 0,C 180,E1 -26617.941,E2 -26617.941} C_VEL
LIN {X 0,Y 188.939,Z 271.235,A -85,B 0,C 180,E1 -26620.723,E2 -26620.723} C_VEL
LIN {X 0,Y 186.434,Z 265.996,A -85,B 0,C 180,E1 -26623.788,E2 -26623.788} C_VEL
LIN {X 0,Y 184.009,Z 261.064,A -85,B 0,C 180,E1 -26627.524,E2 -26627.524} C_VEL
LIN {X 0,Y 182.199,Z 257.396,A -85,B 0,C 180,E1 -26631.403,E2 -26631.403} C_VEL
LIN {X 0,Y 180.838,Z 253.419,A -85,B 0,C 180,E1 -26637.772,E2 -26637.772} C_VEL
LIN {X 0,Y 180.846,Z 253.423,A -85,B 0,C 180,E1 -26641.948,E2 -26641.948} C_VEL
LIN {X 0,Y 182.229,Z 257.409,A -85,B 0,C 180,E1 -26648.315,E2 -26648.315} C_VEL
LIN {X 0,Y 184.319,Z 261.658,A -85,B 0,C 180,E1 -26652.664,E2 -26652.664} C_VEL
LIN {X 0,Y 186.661,Z 266.383,A -85,B 0,C 180,E1 -26656.155,E2 -26656.155} C_VEL
LIN {X 0,Y 189.039,Z 271.573,A -85,B 0,C 180,E1 -26659.054,E2 -26659.054} C_VEL
LIN {X 0,Y 191.237,Z 278.518,A -85,B 0,C 180,E1 -26661.561,E2 -26661.561} C_VEL
LIN {X 0,Y 191.474,Z 279.304,A -85,B 0,C 180,E1 -26661.816,E2 -26661.816} C_VEL
LIN {X 0,Y 186.846,Z 323.955,A -85,B 0,C 180,E1 -26662.952,E2 -26662.952} C_VEL
LIN {X 0,Y 183.946,Z 339.289,A -85,B 0,C 180,E1 -26663.513,E2 -26663.513} C_VEL
LIN {X 0,Y 179.793,Z 354.502,A -85,B 0,C 180,E1 -26664.317,E2 -26664.317} C_VEL
LIN {X 0,Y 174.919,Z 368.219,A -85,B 0,C 180,E1 -26665.308,E2 -26665.308} C_VEL
LIN {X 0,Y 169.015,Z 381.66,A -85,B 0,C 180,E1 -26666.617,E2 -26666.617} C_VEL
LIN {X 0,Y 161.874,Z 395.361,A -85,B 0,C 180,E1 -26668.458,E2 -26668.458} C_VEL
LIN {X 0,Y 154.235,Z 407.764,A -85,B 0,C 180,E1 -26670.674,E2 -26670.674} C_VEL
LIN {X 0,Y 145.443,Z 419.926,A -85,B 0,C 180,E1 -26673.535,E2 -26673.535} C_VEL
LIN {X 0,Y 136.528,Z 430.756,A -85,B 0,C 180,E1 -26677.071,E2 -26677.071} C_VEL
LIN {X 0,Y 128.342,Z 439.715,A -85,B 0,C 180,E1 -26681.08,E2 -26681.08} C_VEL
LIN {X 0,Y 120.864,Z 447.29,A -85,B 0,C 180,E1 -26685.751,E2 -26685.751} C_VEL
LIN {X 0,Y 113.201,Z 454.285,A -85,B 0,C 180,E1 -26691.622,E2 -26691.622} C_VEL
LIN {X 0,Y 106.329,Z 460.444,A -85,B 0,C 180,E1 -26699.232,E2 -26699.232} C_VEL
LIN {X 0,Y 102.354,Z 463.975,A -85,B 0,C 180,E1 -26705.67,E2 -26705.67} C_VEL
LIN {X 0,Y 99.3,Z 466.911,A -85,B 0,C 180,E1 -26713.554,E2 -26713.554} C_VEL
LIN {X 0,Y 98.006,Z 468.673,A -85,B 0,C 180,E1 -26721.754,E2 -26721.754} C_VEL
LIN {X 0,Y 98.071,Z 469.286,A -85,B 0,C 180,E1 -26730,E2 -26730} C_VEL
LIN {X 0,Y 98.004,Z 468.653,A -85,B 0,C 180,E1 -26738.246,E2 -26738.246} C_VEL
LIN {X 0,Y 99.285,Z 466.863,A -85,B 0,C 180,E1 -26746.448,E2 -26746.448} C_VEL
LIN {X 0,Y 99.638,Z 466.442,A -85,B 0,C 180,E1 -26747.725,E2 -26747.725} C_VEL
LIN {X 0,Y 100.097,Z 465.357,A -85,B 0,C 180,E1 -26751.041,E2 -26751.041} C_VEL
LIN {X 0,Y 99.742,Z 463.16,A -85,B 0,C 180,E1 -26756.592,E2 -26756.592} C_VEL
LIN {X 0,Y 99.952,Z 461.091,A -85,B 0,C 180,E1 -26761.004,E2 -26761.004} C_VEL
LIN {X 0,Y 101.233,Z 459.305,A -85,B 0,C 180,E1 -26764.135,E2 -26764.135} C_VEL
LIN {X 0,Y 101.971,Z 458.641,A -85,B 0,C 180,E1 -26765.102,E2 -26765.102} C_VEL
LIN {X 0,Y 109.528,Z 452.329,A -85,B 0,C 180,E1 -26772.357,E2 -26772.357} C_VEL
LIN {X 0,Y 117.944,Z 444.89,A -85,B 0,C 180,E1 -26778.146,E2 -26778.146} C_VEL
LIN {X 0,Y 126.039,Z 436.932,A -85,B 0,C 180,E1 -26782.616,E2 -26782.616} C_VEL
LIN {X 0,Y 134.924,Z 427.394,A -85,B 0,C 180,E1 -26786.451,E2 -26786.451} C_VEL
LIN {X 0,Y 142.961,Z 417.679,A -85,B 0,C 180,E1 -26789.351,E2 -26789.351} C_VEL
LIN {X 0,Y 151.42,Z 406.154,A -85,B 0,C 180,E1 -26791.869,E2 -26791.869} C_VEL
LIN {X 0,Y 158.591,Z 394.751,A -85,B 0,C 180,E1 -26793.817,E2 -26793.817} C_VEL
LIN {X 0,Y 165.203,Z 382.49,A -85,B 0,C 180,E1 -26795.413,E2 -26795.413} C_VEL
LIN {X 0,Y 171.218,Z 369.226,A -85,B 0,C 180,E1 -26796.698,E2 -26796.698} C_VEL
LIN {X 0,Y 176.583,Z 354.705,A -85,B 0,C 180,E1 -26797.722,E2 -26797.722} C_VEL
LIN {X 0,Y 180.818,Z 339.634,A -85,B 0,C 180,E1 -26798.498,E2 -26798.498} C_VEL
LIN {X 0,Y 183.741,Z 324.674,A -85,B 0,C 180,E1 -26799.045,E2 -26799.045} C_VEL
LIN {X 0,Y 187.044,Z 295.183,A -85,B 0,C 180,E1 -26799.765,E2 -26799.765} C_VEL
LIN {X 0,Y 188.346,Z 282.194,A -85,B 0,C 180,E1 -26800.094,E2 -26800.094} C_VEL
LIN {X 0,Y 186.475,Z 276.204,A -85,B 0,C 180,E1 -26802.452,E2 -26802.452} C_VEL
LIN {X 0,Y 183.982,Z 270.588,A -85,B 0,C 180,E1 -26805.906,E2 -26805.906} C_VEL
LIN {X 0,Y 182.185,Z 266.965,A -85,B 0,C 180,E1 -26809.02,E2 -26809.02} C_VEL
LIN {X 0,Y 180.959,Z 264.175,A -85,B 0,C 180,E1 -26811.907,E2 -26811.907} C_VEL
LIN {X 0,Y 179.688,Z 260.55,A -85,B 0,C 180,E1 -26817.619,E2 -26817.619} C_VEL
LIN {X 0,Y 179.561,Z 260.263,A -85,B 0,C 180,E1 -26821.122,E2 -26821.122} C_VEL
LIN {X 0,Y 179.713,Z 260.853,A -85,B 0,C 180,E1 -26823.223,E2 -26823.223} C_VEL
LIN {X 0,Y 180.946,Z 264.221,A -85,B 0,C 180,E1 -26828.516,E2 -26828.516} C_VEL
LIN {X 0,Y 182.835,Z 268.358,A -85,B 0,C 180,E1 -26832.656,E2 -26832.656} C_VEL
LIN {X 0,Y 184.578,Z 272.076,A -85,B 0,C 180,E1 -26835.458,E2 -26835.458} C_VEL
LIN {X 0,Y 187.357,Z 278.295,A -85,B 0,C 180,E1 -26839.055,E2 -26839.055} C_VEL
LIN {X 0,Y 188.408,Z 280.84,A -85,B 0,C 180,E1 -26840.25,E2 -26840.25} C_VEL
LIN {X 0,Y 184.33,Z 319.511,A -85,B 0,C 180,E1 -26841.235,E2 -26841.235} C_VEL
LIN {X 0,Y 181.433,Z 334.942,A -85,B 0,C 180,E1 -26841.805,E2 -26841.805} C_VEL
LIN {X 0,Y 177.114,Z 350.781,A -85,B 0,C 180,E1 -26842.694,E2 -26842.694} C_VEL
LIN {X 0,Y 171.94,Z 365.274,A -85,B 0,C 180,E1 -26843.854,E2 -26843.854} C_VEL
LIN {X 0,Y 165.709,Z 379.34,A -85,B 0,C 180,E1 -26845.393,E2 -26845.393} C_VEL
LIN {X 0,Y 158.928,Z 391.922,A -85,B 0,C 180,E1 -26847.132,E2 -26847.132} C_VEL
LIN {X 0,Y 151.109,Z 404.122,A -85,B 0,C 180,E1 -26849.302,E2 -26849.302} C_VEL
LIN {X 0,Y 142.907,Z 415.234,A -85,B 0,C 180,E1 -26851.969,E2 -26851.969} C_VEL
LIN {X 0,Y 134.568,Z 425.038,A -85,B 0,C 180,E1 -26855.064,E2 -26855.064} C_VEL
LIN {X 0,Y 126.495,Z 433.751,A -85,B 0,C 180,E1 -26858.937,E2 -26858.937} C_VEL
LIN {X 0,Y 118.418,Z 441.382,A -85,B 0,C 180,E1 -26863.362,E2 -26863.362} C_VEL
LIN {X 0,Y 111.147,Z 447.706,A -85,B 0,C 180,E1 -26868.4,E2 -26868.4} C_VEL
LIN {X 0,Y 104.007,Z 453.509,A -85,B 0,C 180,E1 -26874.945,E2 -26874.945} C_VEL
LIN {X 0,Y 99.646,Z 456.938,A -85,B 0,C 180,E1 -26880.415,E2 -26880.415} C_VEL
LIN {X 0,Y 95.123,Z 460.404,A -85,B 0,C 180,E1 -26888.321,E2 -26888.321} C_VEL
LIN {X 0,Y 92.315,Z 462.685,A -85,B 0,C 180,E1 -26896.798,E2 -26896.798} C_VEL
LIN {X 0,Y 91.106,Z 463.839,A -85,B 0,C 180,E1 -26905.576,E2 -26905.576} C_VEL
LIN {X 0,Y 91.056,Z 463.99,A -85,B 0,C 180,E1 -26910,E2 -26910} C_VEL
LIN {X 0,Y 91.542,Z 463.43,A -85,B 0,C 180,E1 -26918.833,E2 -26918.833} C_VEL
LIN {X 0,Y 93.476,Z 461.76,A -85,B 0,C 180,E1 -26927.502,E2 -26927.502} C_VEL
LIN {X 0,Y 97.067,Z 458.934,A -85,B 0,C 180,E1 -26935.749,E2 -26935.749} C_VEL
LIN {X 0,Y 102.403,Z 454.877,A -85,B 0,C 180,E1 -26943.302,E2 -26943.302} C_VEL
LIN {X 0,Y 109.176,Z 449.492,A -85,B 0,C 180,E1 -26950.071,E2 -26950.071} C_VEL
LIN {X 0,Y 117.248,Z 442.623,A -85,B 0,C 180,E1 -26955.997,E2 -26955.997} C_VEL
LIN {X 0,Y 125.205,Z 435.236,A -85,B 0,C 180,E1 -26960.518,E2 -26960.518} C_VEL
LIN {X 0,Y 133.493,Z 426.582,A -85,B 0,C 180,E1 -26964.444,E2 -26964.444} C_VEL
LIN {X 0,Y 141.464,Z 417.239,A -85,B 0,C 180,E1 -26967.626,E2 -26967.626} C_VEL
LIN {X 0,Y 149.647,Z 406.508,A -85,B 0,C 180,E1 -26970.324,E2 -26970.324} C_VEL
LIN {X 0,Y 157.39,Z 394.788,A -85,B 0,C 180,E1 -26972.56,E2 -26972.56} C_VEL
LIN {X 0,Y 164.388,Z 382.376,A -85,B 0,C 180,E1 -26974.379,E2 -26974.379} C_VEL
LIN {X 0,Y 170.371,Z 369.607,A -85,B 0,C 180,E1 -26975.88,E2 -26975.88} C_VEL
LIN {X 0,Y 175.936,Z 355.175,A -85,B 0,C 180,E1 -26977.113,E2 -26977.113} C_VEL
LIN {X 0,Y 180.238,Z 340.87,A -85,B 0,C 180,E1 -26978.019,E2 -26978.019} C_VEL
LIN {X 0,Y 183.619,Z 325.465,A -85,B 0,C 180,E1 -26978.69,E2 -26978.69} C_VEL
LIN {X 0,Y 185.799,Z 309.373,A -85,B 0,C 180,E1 -26979.167,E2 -26979.167} C_VEL
LIN {X 0,Y 188.666,Z 281.017,A -85,B 0,C 180,E1 -26979.866,E2 -26979.866} C_VEL
LIN {X 0,Y 185.986,Z 274.809,A -85,B 0,C 180,E1 -26983.077,E2 -26983.077} C_VEL
LIN {X 0,Y 183.693,Z 269.864,A -85,B 0,C 180,E1 -26986.44,E2 -26986.44} C_VEL
LIN {X 0,Y 182.357,Z 267.075,A -85,B 0,C 180,E1 -26988.889,E2 -26988.889} C_VEL
LIN {X 0,Y 181.143,Z 264.284,A -85,B 0,C 180,E1 -26991.845,E2 -26991.845} C_VEL
LIN {X 0,Y 179.926,Z 260.412,A -85,B 0,C 180,E1 -26998.321,E2 -26998.321} C_VEL
LIN {X 0,Y 179.949,Z 260.479,A -85,B 0,C 180,E1 -27001.678,E2 -27001.678} C_VEL
LIN {X 0,Y 181.451,Z 264.902,A -85,B 0,C 180,E1 -27008.632,E2 -27008.632} C_VEL
LIN {X 0,Y 183.183,Z 268.723,A -85,B 0,C 180,E1 -27012.322,E2 -27012.322} C_VEL
LIN {X 0,Y 185.331,Z 273.268,A -85,B 0,C 180,E1 -27015.675,E2 -27015.675} C_VEL
LIN {X 0,Y 187.142,Z 277.578,A -85,B 0,C 180,E1 -27018.048,E2 -27018.048} C_VEL
LIN {X 0,Y 188.59,Z 282.469,A -85,B 0,C 180,E1 -27019.88,E2 -27019.88} C_VEL
LIN {X 0,Y 184.309,Z 323.038,A -85,B 0,C 180,E1 -27020.894,E2 -27020.894} C_VEL
LIN {X 0,Y 181.385,Z 338.434,A -85,B 0,C 180,E1 -27021.418,E2 -27021.418} C_VEL
LIN {X 0,Y 176.985,Z 354.31,A -85,B 0,C 180,E1 -27022.22,E2 -27022.22} C_VEL
LIN {X 0,Y 172,Z 368.026,A -85,B 0,C 180,E1 -27023.167,E2 -27023.167} C_VEL
LIN {X 0,Y 165.955,Z 381.466,A -85,B 0,C 180,E1 -27024.425,E2 -27024.425} C_VEL
LIN {X 0,Y 159.051,Z 394.373,A -85,B 0,C 180,E1 -27026.082,E2 -27026.082} C_VEL
LIN {X 0,Y 151.433,Z 406.496,A -85,B 0,C 180,E1 -27028.141,E2 -27028.141} C_VEL
LIN {X 0,Y 142.986,Z 417.969,A -85,B 0,C 180,E1 -27030.666,E2 -27030.666} C_VEL
LIN {X 0,Y 134.945,Z 427.633,A -85,B 0,C 180,E1 -27033.561,E2 -27033.561} C_VEL
LIN {X 0,Y 126.078,Z 437.133,A -85,B 0,C 180,E1 -27037.406,E2 -27037.406} C_VEL
LIN {X 0,Y 118.01,Z 445.059,A -85,B 0,C 180,E1 -27041.889,E2 -27041.889} C_VEL
LIN {X 0,Y 109.574,Z 452.459,A -85,B 0,C 180,E1 -27047.665,E2 -27047.665} C_VEL
LIN {X 0,Y 102.507,Z 458.341,A -85,B 0,C 180,E1 -27054.354,E2 -27054.354} C_VEL
LIN {X 0,Y 98.239,Z 461.847,A -85,B 0,C 180,E1 -27059.948,E2 -27059.948} C_VEL
LIN {X 0,Y 93.931,Z 465.393,A -85,B 0,C 180,E1 -27068.031,E2 -27068.031} C_VEL
LIN {X 0,Y 91.502,Z 467.737,A -85,B 0,C 180,E1 -27076.678,E2 -27076.678} C_VEL
LIN {X 0,Y 90.807,Z 468.925,A -85,B 0,C 180,E1 -27085.561,E2 -27085.561} C_VEL
LIN {X 0,Y 90.969,Z 469.087,A -85,B 0,C 180,E1 -27090,E2 -27090} C_VEL
LIN {X 0,Y 90.95,Z 468.453,A -85,B 0,C 180,E1 -27098.89,E2 -27098.89} C_VEL
LIN {X 0,Y 92.655,Z 466.425,A -85,B 0,C 180,E1 -27108.474,E2 -27108.474} C_VEL
LIN {X 0,Y 95.801,Z 463.701,A -85,B 0,C 180,E1 -27116.114,E2 -27116.114} C_VEL
LIN {X 0,Y 100.912,Z 459.503,A -85,B 0,C 180,E1 -27123.859,E2 -27123.859} C_VEL
LIN {X 0,Y 101.971,Z 458.641,A -85,B 0,C 180,E1 -27125.102,E2 -27125.102} C_VEL
LIN {X 0,Y 103.968,Z 456.632,A -85,B 0,C 180,E1 -27127.979,E2 -27127.979} C_VEL
LIN {X 0,Y 106.18,Z 453.06,A -85,B 0,C 180,E1 -27132.867,E2 -27132.867} C_VEL
LIN {X 0,Y 108.9,Z 449,A -85,B 0,C 180,E1 -27137.465,E2 -27137.465} C_VEL
LIN {X 0,Y 111.577,Z 446.215,A -85,B 0,C 180,E1 -27139.792,E2 -27139.792} C_VEL
LIN {X 0,Y 120.56,Z 437.969,A -85,B 0,C 180,E1 -27144.699,E2 -27144.699} C_VEL
LIN {X 0,Y 129.744,Z 428.684,A -85,B 0,C 180,E1 -27148.556,E2 -27148.556} C_VEL
LIN {X 0,Y 138.044,Z 419.255,A -85,B 0,C 180,E1 -27151.428,E2 -27151.428} C_VEL
LIN {X 0,Y 147.467,Z 407.024,A -85,B 0,C 180,E1 -27154.099,E2 -27154.099} C_VEL
LIN {X 0,Y 155.578,Z 394.548,A -85,B 0,C 180,E1 -27156.172,E2 -27156.172} C_VEL
LIN {X 0,Y 162.375,Z 382.287,A -85,B 0,C 180,E1 -27157.693,E2 -27157.693} C_VEL
LIN {X 0,Y 168.527,Z 369.021,A -85,B 0,C 180,E1 -27158.922,E2 -27158.922} C_VEL
LIN {X 0,Y 174.01,Z 354.499,A -85,B 0,C 180,E1 -27159.89,E2 -27159.89} C_VEL
LIN {X 0,Y 178.338,Z 339.426,A -85,B 0,C 180,E1 -27160.62,E2 -27160.62} C_VEL
LIN {X 0,Y 181.181,Z 325.269,A -85,B 0,C 180,E1 -27161.12,E2 -27161.12} C_VEL
LIN {X 0,Y 184.083,Z 300.798,A -85,B 0,C 180,E1 -27161.711,E2 -27161.711} C_VEL
LIN {X 0,Y 185.65,Z 285.548,A -85,B 0,C 180,E1 -27162.09,E2 -27162.09} C_VEL
LIN {X 0,Y 184.57,Z 281.992,A -85,B 0,C 180,E1 -27163.611,E2 -27163.611} C_VEL
LIN {X 0,Y 182.399,Z 276.822,A -85,B 0,C 180,E1 -27166.917,E2 -27166.917} C_VEL
LIN {X 0,Y 180.896,Z 273.547,A -85,B 0,C 180,E1 -27169.79,E2 -27169.79} C_VEL
LIN {X 0,Y 179.88,Z 271.026,A -85,B 0,C 180,E1 -27172.423,E2 -27172.423} C_VEL
LIN {X 0,Y 178.762,Z 267.395,A -85,B 0,C 180,E1 -27178.311,E2 -27178.311} C_VEL
LIN {X 0,Y 178.696,Z 267.303,A -85,B 0,C 180,E1 -27181.127,E2 -27181.127} C_VEL
LIN {X 0,Y 178.802,Z 267.759,A -85,B 0,C 180,E1 -27182.816,E2 -27182.816} C_VEL
LIN {X 0,Y 179.82,Z 270.978,A -85,B 0,C 180,E1 -27187.863,E2 -27187.863} C_VEL
LIN {X 0,Y 181.595,Z 275.146,A -85,B 0,C 180,E1 -27192.09,E2 -27192.09} C_VEL
LIN {X 0,Y 183.304,Z 278.985,A -85,B 0,C 180,E1 -27194.999,E2 -27194.999} C_VEL
LIN {X 0,Y 185.694,Z 284.816,A -85,B 0,C 180,E1 -27198.301,E2 -27198.301} C_VEL
LIN {X 0,Y 181.782,Z 320.369,A -85,B 0,C 180,E1 -27199.179,E2 -27199.179} C_VEL
LIN {X 0,Y 178.916,Z 335.151,A -85,B 0,C 180,E1 -27199.692,E2 -27199.692} C_VEL
LIN {X 0,Y 174.504,Z 350.987,A -85,B 0,C 180,E1 -27200.548,E2 -27200.548} C_VEL
LIN {X 0,Y 169.191,Z 365.479,A -85,B 0,C 180,E1 -27201.653,E2 -27201.653} C_VEL
LIN {X 0,Y 162.651,Z 379.8,A -85,B 0,C 180,E1 -27203.162,E2 -27203.162} C_VEL
LIN {X 0,Y 155.815,Z 392.125,A -85,B 0,C 180,E1 -27204.806,E2 -27204.806} C_VEL
LIN {X 0,Y 147.761,Z 404.324,A -85,B 0,C 180,E1 -27206.898,E2 -27206.898} C_VEL
LIN {X 0,Y 139.281,Z 415.436,A -85,B 0,C 180,E1 -27209.492,E2 -27209.492} C_VEL
LIN {X 0,Y 130.195,Z 425.699,A -85,B 0,C 180,E1 -27212.671,E2 -27212.671} C_VEL
LIN {X 0,Y 122.157,Z 433.952,A -85,B 0,C 180,E1 -27216.346,E2 -27216.346} C_VEL
LIN {X 0,Y 113.646,Z 441.583,A -85,B 0,C 180,E1 -27220.751,E2 -27220.751} C_VEL
LIN {X 0,Y 105.925,Z 447.907,A -85,B 0,C 180,E1 -27225.84,E2 -27225.84} C_VEL
LIN {X 0,Y 98.251,Z 453.709,A -85,B 0,C 180,E1 -27232.554,E2 -27232.554} C_VEL
LIN {X 0,Y 93.505,Z 457.139,A -85,B 0,C 180,E1 -27238.256,E2 -27238.256} C_VEL
LIN {X 0,Y 88.53,Z 460.605,A -85,B 0,C 180,E1 -27246.614,E2 -27246.614} C_VEL
LIN {X 0,Y 85.411,Z 462.884,A -85,B 0,C 180,E1 -27255.709,E2 -27255.709} C_VEL
LIN {X 0,Y 84.05,Z 464.037,A -85,B 0,C 180,E1 -27265.204,E2 -27265.204} C_VEL
LIN {X 0,Y 83.956,Z 464.189,A -85,B 0,C 180,E1 -27270,E2 -27270} C_VEL
LIN {X 0,Y 84.514,Z 463.629,A -85,B 0,C 180,E1 -27279.574,E2 -27279.574} C_VEL
LIN {X 0,Y 86.704,Z 461.959,A -85,B 0,C 180,E1 -27288.919,E2 -27288.919} C_VEL
LIN {X 0,Y 90.694,Z 459.133,A -85,B 0,C 180,E1 -27297.707,E2 -27297.707} C_VEL
LIN {X 0,Y 96.509,Z 455.076,A -85,B 0,C 180,E1 -27305.632,E2 -27305.632} C_VEL
LIN {X 0,Y 103.811,Z 449.691,A -85,B 0,C 180,E1 -27312.61,E2 -27312.61} C_VEL
LIN {X 0,Y 112.409,Z 442.821,A -85,B 0,C 180,E1 -27318.613,E2 -27318.613} C_VEL
LIN {X 0,Y 120.812,Z 435.433,A -85,B 0,C 180,E1 -27323.119,E2 -27323.119} C_VEL
LIN {X 0,Y 129.024,Z 427.244,A -85,B 0,C 180,E1 -27326.827,E2 -27326.827} C_VEL
LIN {X 0,Y 137.793,Z 417.435,A -85,B 0,C 180,E1 -27330.12,E2 -27330.12} C_VEL
LIN {X 0,Y 146.258,Z 406.704,A -85,B 0,C 180,E1 -27332.744,E2 -27332.744} C_VEL
LIN {X 0,Y 154.242,Z 394.984,A -85,B 0,C 180,E1 -27334.905,E2 -27334.905} C_VEL
LIN {X 0,Y 160.917,Z 383.597,A -85,B 0,C 180,E1 -27336.517,E2 -27336.517} C_VEL
LIN {X 0,Y 166.848,Z 371.546,A -85,B 0,C 180,E1 -27337.925,E2 -27337.925} C_VEL
LIN {X 0,Y 172.529,Z 357.576,A -85,B 0,C 180,E1 -27339.126,E2 -27339.126} C_VEL
LIN {X 0,Y 177.146,Z 343.209,A -85,B 0,C 180,E1 -27340.013,E2 -27340.013} C_VEL
LIN {X 0,Y 180.846,Z 327.483,A -85,B 0,C 180,E1 -27340.712,E2 -27340.712} C_VEL
LIN {X 0,Y 183.256,Z 310.983,A -85,B 0,C 180,E1 -27341.196,E2 -27341.196} C_VEL
LIN {X 0,Y 185.9,Z 284.863,A -85,B 0,C 180,E1 -27341.885,E2 -27341.885} C_VEL
LIN {X 0,Y 183.545,Z 279.233,A -85,B 0,C 180,E1 -27345.145,E2 -27345.145} C_VEL
LIN {X 0,Y 181.609,Z 274.696,A -85,B 0,C 180,E1 -27348.56,E2 -27348.56} C_VEL
LIN {X 0,Y 180.05,Z 271.097,A -85,B 0,C 180,E1 -27352.43,E2 -27352.43} C_VEL
LIN {X 0,Y 179.061,Z 267.452,A -85,B 0,C 180,E1 -27358.313,E2 -27358.313} C_VEL
LIN {X 0,Y 179.062,Z 267.596,A -85,B 0,C 180,E1 -27361.546,E2 -27361.546} C_VEL
LIN {X 0,Y 180.359,Z 271.739,A -85,B 0,C 180,E1 -27368.12,E2 -27368.12} C_VEL
LIN {X 0,Y 181.967,Z 275.553,A -85,B 0,C 180,E1 -27371.805,E2 -27371.805} C_VEL
LIN {X 0,Y 183.891,Z 279.968,A -85,B 0,C 180,E1 -27375.02,E2 -27375.02} C_VEL
LIN {X 0,Y 185.351,Z 283.728,A -85,B 0,C 180,E1 -27377.089,E2 -27377.089} C_VEL
LIN {X 0,Y 185.907,Z 285.784,A -85,B 0,C 180,E1 -27377.885,E2 -27377.885} C_VEL
LIN {X 0,Y 181.79,Z 323.515,A -85,B 0,C 180,E1 -27378.824,E2 -27378.824} C_VEL
LIN {X 0,Y 178.881,Z 338.349,A -85,B 0,C 180,E1 -27379.298,E2 -27379.298} C_VEL
LIN {X 0,Y 174.42,Z 354.118,A -85,B 0,C 180,E1 -27380.058,E2 -27380.058} C_VEL
LIN {X 0,Y 169.327,Z 367.833,A -85,B 0,C 180,E1 -27380.952,E2 -27380.952} C_VEL
LIN {X 0,Y 163.143,Z 381.272,A -85,B 0,C 180,E1 -27382.15,E2 -27382.15} C_VEL
LIN {X 0,Y 155.587,Z 394.964,A -85,B 0,C 180,E1 -27383.834,E2 -27383.834} C_VEL
LIN {X 0,Y 147.47,Z 407.371,A -85,B 0,C 180,E1 -27385.903,E2 -27385.903} C_VEL
LIN {X 0,Y 138.069,Z 419.531,A -85,B 0,C 180,E1 -27388.59,E2 -27388.59} C_VEL
LIN {X 0,Y 128.412,Z 430.359,A -85,B 0,C 180,E1 -27391.97,E2 -27391.97} C_VEL
LIN {X 0,Y 119.376,Z 439.352,A -85,B 0,C 180,E1 -27395.907,E2 -27395.907} C_VEL
LIN {X 0,Y 111.059,Z 446.892,A -85,B 0,C 180,E1 -27400.59,E2 -27400.59} C_VEL
LIN {X 0,Y 102.349,Z 453.886,A -85,B 0,C 180,E1 -27406.632,E2 -27406.632} C_VEL
LIN {X 0,Y 95.093,Z 459.398,A -85,B 0,C 180,E1 -27413.754,E2 -27413.754} C_VEL
LIN {X 0,Y 89.469,Z 463.574,A -85,B 0,C 180,E1 -27421.88,E2 -27421.88} C_VEL
LIN {X 0,Y 85.649,Z 466.51,A -85,B 0,C 180,E1 -27430.839,E2 -27430.839} C_VEL
LIN {X 0,Y 83.9,Z 468.274,A -85,B 0,C 180,E1 -27440.355,E2 -27440.355} C_VEL
LIN {X 0,Y 83.875,Z 468.888,A -85,B 0,C 180,E1 -27450,E2 -27450} C_VEL
LIN {X 0,Y 83.728,Z 468.72,A -85,B 0,C 180,E1 -27454.815,E2 -27454.815} C_VEL
LIN {X 0,Y 84.552,Z 467.501,A -85,B 0,C 180,E1 -27464.44,E2 -27464.44} C_VEL
LIN {X 0,Y 87.29,Z 465.13,A -85,B 0,C 180,E1 -27473.738,E2 -27473.738} C_VEL
LIN {X 0,Y 91.987,Z 461.56,A -85,B 0,C 180,E1 -27482.331,E2 -27482.331} C_VEL
LIN {X 0,Y 98.494,Z 456.706,A -85,B 0,C 180,E1 -27489.955,E2 -27489.955} C_VEL
LIN {X 0,Y 106.482,Z 450.436,A -85,B 0,C 180,E1 -27496.554,E2 -27496.554} C_VEL
LIN {X 0,Y 111.577,Z 446.215,A -85,B 0,C 180,E1 -27499.792,E2 -27499.792} C_VEL
LIN {X 0,Y 114.365,Z 443.352,A -85,B 0,C 180,E1 -27501.99,E2 -27501.99} C_VEL
LIN {X 0,Y 121.023,Z 434.25,A -85,B 0,C 180,E1 -27508.747,E2 -27508.747} C_VEL
LIN {X 0,Y 123.965,Z 430.783,A -85,B 0,C 180,E1 -27510.5,E2 -27510.5} C_VEL
LIN {X 0,Y 125.12,Z 429.555,A -85,B 0,C 180,E1 -27510.964,E2 -27510.964} C_VEL
LIN {X 0,Y 134.77,Z 419.052,A -85,B 0,C 180,E1 -27514.1,E2 -27514.1} C_VEL
LIN {X 0,Y 144.484,Z 406.82,A -85,B 0,C 180,E1 -27516.653,E2 -27516.653} C_VEL
LIN {X 0,Y 152.833,Z 394.344,A -85,B 0,C 180,E1 -27518.622,E2 -27518.622} C_VEL
LIN {X 0,Y 159.813,Z 382.083,A -85,B 0,C 180,E1 -27520.051,E2 -27520.051} C_VEL
LIN {X 0,Y 166.099,Z 368.816,A -85,B 0,C 180,E1 -27521.216,E2 -27521.216} C_VEL
LIN {X 0,Y 171.695,Z 354.293,A -85,B 0,C 180,E1 -27522.119,E2 -27522.119} C_VEL
LIN {X 0,Y 176.11,Z 339.218,A -85,B 0,C 180,E1 -27522.799,E2 -27522.799} C_VEL
LIN {X 0,Y 179.152,Z 324.26,A -85,B 0,C 180,E1 -27523.29,E2 -27523.29} C_VEL
LIN {X 0,Y 182.54,Z 295.502,A -85,B 0,C 180,E1 -27523.929,E2 -27523.929} C_VEL
LIN {X 0,Y 183.192,Z 289.146,A -85,B 0,C 180,E1 -27524.102,E2 -27524.102} C_VEL
LIN {X 0,Y 181.554,Z 284.746,A -85,B 0,C 180,E1 -27526.712,E2 -27526.712} C_VEL
LIN {X 0,Y 179.886,Z 280.597,A -85,B 0,C 180,E1 -27530.016,E2 -27530.016} C_VEL
LIN {X 0,Y 178.79,Z 277.855,A -85,B 0,C 180,E1 -27533.015,E2 -27533.015} C_VEL
LIN {X 0,Y 177.891,Z 274.494,A -85,B 0,C 180,E1 -27538.302,E2 -27538.302} C_VEL
LIN {X 0,Y 177.861,Z 274.406,A -85,B 0,C 180,E1 -27541.698,E2 -27541.698} C_VEL
LIN {X 0,Y 179.024,Z 278.512,A -85,B 0,C 180,E1 -27548.182,E2 -27548.182} C_VEL
LIN {X 0,Y 180.439,Z 282.074,A -85,B 0,C 180,E1 -27551.65,E2 -27551.65} C_VEL
LIN {X 0,Y 182.075,Z 286.078,A -85,B 0,C 180,E1 -27554.602,E2 -27554.602} C_VEL
LIN {X 0,Y 183.152,Z 288.903,A -85,B 0,C 180,E1 -27556.259,E2 -27556.259} C_VEL
LIN {X 0,Y 179.546,Z 320.756,A -85,B 0,C 180,E1 -27557.045,E2 -27557.045} C_VEL
LIN {X 0,Y 176.462,Z 336.125,A -85,B 0,C 180,E1 -27557.566,E2 -27557.566} C_VEL
LIN {X 0,Y 172.145,Z 351.192,A -85,B 0,C 180,E1 -27558.339,E2 -27558.339} C_VEL
LIN {X 0,Y 166.704,Z 365.683,A -85,B 0,C 180,E1 -27559.386,E2 -27559.386} C_VEL
LIN {X 0,Y 160.359,Z 379.289,A -85,B 0,C 180,E1 -27560.724,E2 -27560.724} C_VEL
LIN {X 0,Y 152.973,Z 392.327,A -85,B 0,C 180,E1 -27562.391,E2 -27562.391} C_VEL
LIN {X 0,Y 144.673,Z 404.527,A -85,B 0,C 180,E1 -27564.377,E2 -27564.377} C_VEL
LIN {X 0,Y 135.919,Z 415.638,A -85,B 0,C 180,E1 -27566.88,E2 -27566.88} C_VEL
LIN {X 0,Y 126.081,Z 426.322,A -85,B 0,C 180,E1 -27570.111,E2 -27570.111} C_VEL
LIN {X 0,Y 116.742,Z 435.368,A -85,B 0,C 180,E1 -27574.13,E2 -27574.13} C_VEL
LIN {X 0,Y 107.901,Z 442.784,A -85,B 0,C 180,E1 -27578.592,E2 -27578.592} C_VEL
LIN {X 0,Y 98.738,Z 449.707,A -85,B 0,C 180,E1 -27584.62,E2 -27584.62} C_VEL
LIN {X 0,Y 90.842,Z 455.137,A -85,B 0,C 180,E1 -27591.763,E2 -27591.763} C_VEL
LIN {X 0,Y 84.489,Z 459.227,A -85,B 0,C 180,E1 -27600.06,E2 -27600.06} C_VEL
LIN {X 0,Y 80.054,Z 462.087,A -85,B 0,C 180,E1 -27609.442,E2 -27609.442} C_VEL
LIN {X 0,Y 77.513,Z 463.798,A -85,B 0,C 180,E1 -27619.553,E2 -27619.553} C_VEL
LIN {X 0,Y 76.883,Z 464.387,A -85,B 0,C 180,E1 -27630,E2 -27630} C_VEL
LIN {X 0,Y 77.511,Z 463.828,A -85,B 0,C 180,E1 -27640.448,E2 -27640.448} C_VEL
LIN {X 0,Y 80.003,Z 462.158,A -85,B 0,C 180,E1 -27650.572,E2 -27650.572} C_VEL
LIN {X 0,Y 84.447,Z 459.332,A -85,B 0,C 180,E1 -27659.957,E2 -27659.957} C_VEL
LIN {X 0,Y 90.802,Z 455.275,A -85,B 0,C 180,E1 -27668.258,E2 -27668.258} C_VEL
LIN {X 0,Y 98.675,Z 449.89,A -85,B 0,C 180,E1 -27675.418,E2 -27675.418} C_VEL
LIN {X 0,Y 107.829,Z 443.019,A -85,B 0,C 180,E1 -27681.456,E2 -27681.456} C_VEL
LIN {X 0,Y 116.682,Z 435.63,A -85,B 0,C 180,E1 -27685.914,E2 -27685.914} C_VEL
LIN {X 0,Y 126.038,Z 426.661,A -85,B 0,C 180,E1 -27689.877,E2 -27689.877} C_VEL
LIN {X 0,Y 134.39,Z 417.632,A -85,B 0,C 180,E1 -27692.752,E2 -27692.752} C_VEL
LIN {X 0,Y 143.137,Z 406.9,A -85,B 0,C 180,E1 -27695.279,E2 -27695.279} C_VEL
LIN {X 0,Y 151.371,Z 395.178,A -85,B 0,C 180,E1 -27697.337,E2 -27697.337} C_VEL
LIN {X 0,Y 158.98,Z 382.367,A -85,B 0,C 180,E1 -27699.05,E2 -27699.05} C_VEL
LIN {X 0,Y 165.074,Z 369.994,A -85,B 0,C 180,E1 -27700.386,E2 -27700.386} C_VEL
LIN {X 0,Y 170.924,Z 355.557,A -85,B 0,C 180,E1 -27701.493,E2 -27701.493} C_VEL
LIN {X 0,Y 175.425,Z 341.247,A -85,B 0,C 180,E1 -27702.316,E2 -27702.316} C_VEL
LIN {X 0,Y 178.811,Z 326.698,A -85,B 0,C 180,E1 -27702.89,E2 -27702.89} C_VEL
LIN {X 0,Y 181.192,Z 310.193,A -85,B 0,C 180,E1 -27703.349,E2 -27703.349} C_VEL
LIN {X 0,Y 183.412,Z 289.059,A -85,B 0,C 180,E1 -27703.87,E2 -27703.87} C_VEL
LIN {X 0,Y 181.298,Z 283.682,A -85,B 0,C 180,E1 -27707.334,E2 -27707.334} C_VEL
LIN {X 0,Y 179.838,Z 280.227,A -85,B 0,C 180,E1 -27710.439,E2 -27710.439} C_VEL
LIN {X 0,Y 178.997,Z 277.945,A -85,B 0,C 180,E1 -27712.952,E2 -27712.952} C_VEL
LIN {X 0,Y 178.163,Z 274.462,A -85,B 0,C 180,E1 -27718.87,E2 -27718.87} C_VEL
LIN {X 0,Y 178.175,Z 274.536,A -85,B 0,C 180,E1 -27721.13,E2 -27721.13} C_VEL
LIN {X 0,Y 179.321,Z 278.72,A -85,B 0,C 180,E1 -27727.734,E2 -27727.734} C_VEL
LIN {X 0,Y 180.798,Z 282.48,A -85,B 0,C 180,E1 -27731.349,E2 -27731.349} C_VEL
LIN {X 0,Y 182.478,Z 286.65,A -85,B 0,C 180,E1 -27734.355,E2 -27734.355} C_VEL
LIN {X 0,Y 183.46,Z 289.377,A -85,B 0,C 180,E1 -27735.877,E2 -27735.877} C_VEL
LIN {X 0,Y 179.646,Z 323.18,A -85,B 0,C 180,E1 -27736.67,E2 -27736.67} C_VEL
LIN {X 0,Y 176.523,Z 338.72,A -85,B 0,C 180,E1 -27737.151,E2 -27737.151} C_VEL
LIN {X 0,Y 172.117,Z 353.926,A -85,B 0,C 180,E1 -27737.839,E2 -27737.839} C_VEL
LIN {X 0,Y 166.913,Z 367.639,A -85,B 0,C 180,E1 -27738.668,E2 -27738.668} C_VEL
LIN {X 0,Y 160.59,Z 381.077,A -85,B 0,C 180,E1 -27739.793,E2 -27739.793} C_VEL
LIN {X 0,Y 152.843,Z 394.768,A -85,B 0,C 180,E1 -27741.387,E2 -27741.387} C_VEL
LIN {X 0,Y 144.493,Z 407.174,A -85,B 0,C 180,E1 -27743.355,E2 -27743.355} C_VEL
LIN {X 0,Y 134.791,Z 419.333,A -85,B 0,C 180,E1 -27745.918,E2 -27745.918} C_VEL
LIN {X 0,Y 124.765,Z 430.161,A -85,B 0,C 180,E1 -27749.177,E2 -27749.177} C_VEL
LIN {X 0,Y 116.588,Z 437.974,A -85,B 0,C 180,E1 -27752.442,E2 -27752.442} C_VEL
LIN {X 0,Y 106.533,Z 446.693,A -85,B 0,C 180,E1 -27757.66,E2 -27757.66} C_VEL
LIN {X 0,Y 97.259,Z 453.687,A -85,B 0,C 180,E1 -27763.729,E2 -27763.729} C_VEL
LIN {X 0,Y 89.414,Z 459.198,A -85,B 0,C 180,E1 -27771.037,E2 -27771.037} C_VEL
LIN {X 0,Y 83.212,Z 463.374,A -85,B 0,C 180,E1 -27779.552,E2 -27779.552} C_VEL
LIN {X 0,Y 78.915,Z 466.31,A -85,B 0,C 180,E1 -27789.131,E2 -27789.131} C_VEL
LIN {X 0,Y 76.88,Z 468.075,A -85,B 0,C 180,E1 -27799.465,E2 -27799.465} C_VEL
LIN {X 0,Y 76.771,Z 468.69,A -85,B 0,C 180,E1 -27810,E2 -27810} C_VEL
LIN {X 0,Y 76.878,Z 468.053,A -85,B 0,C 180,E1 -27820.535,E2 -27820.535} C_VEL
LIN {X 0,Y 78.896,Z 466.259,A -85,B 0,C 180,E1 -27830.874,E2 -27830.874} C_VEL
LIN {X 0,Y 83.15,Z 463.298,A -85,B 0,C 180,E1 -27840.473,E2 -27840.473} C_VEL
LIN {X 0,Y 89.348,Z 459.099,A -85,B 0,C 180,E1 -27848.996,E2 -27848.996} C_VEL
LIN {X 0,Y 97.218,Z 453.554,A -85,B 0,C 180,E1 -27856.295,E2 -27856.295} C_VEL
LIN {X 0,Y 106.486,Z 446.519,A -85,B 0,C 180,E1 -27862.372,E2 -27862.372} C_VEL
LIN {X 0,Y 115.351,Z 438.908,A -85,B 0,C 180,E1 -27867.02,E2 -27867.02} C_VEL
LIN {X 0,Y 125.12,Z 429.555,A -85,B 0,C 180,E1 -27870.964,E2 -27870.964} C_VEL
LIN {X 0,Y 128.342,Z 425.873,A -85,B 0,C 180,E1 -27872.43,E2 -27872.43} C_VEL
LIN {X 0,Y 136.048,Z 414.49,A -85,B 0,C 180,E1 -27877.357,E2 -27877.357} C_VEL
LIN {X 0,Y 139.013,Z 410.288,A -85,B 0,C 180,E1 -27878.591,E2 -27878.591} C_VEL
LIN {X 0,Y 140.127,Z 408.821,A -85,B 0,C 180,E1 -27878.898,E2 -27878.898} C_VEL
LIN {X 0,Y 148.805,Z 396.555,A -85,B 0,C 180,E1 -27880.838,E2 -27880.838} C_VEL
LIN {X 0,Y 155.925,Z 384.74,A -85,B 0,C 180,E1 -27882.207,E2 -27882.207} C_VEL
LIN {X 0,Y 163.146,Z 370.381,A -85,B 0,C 180,E1 -27883.433,E2 -27883.433} C_VEL
LIN {X 0,Y 168.841,Z 356.346,A -85,B 0,C 180,E1 -27884.277,E2 -27884.277} C_VEL
LIN {X 0,Y 173.521,Z 341.297,A -85,B 0,C 180,E1 -27884.957,E2 -27884.957} C_VEL
LIN {X 0,Y 176.897,Z 325.96,A -85,B 0,C 180,E1 -27885.443,E2 -27885.443} C_VEL
LIN {X 0,Y 179.618,Z 305.024,A -85,B 0,C 180,E1 -27885.907,E2 -27885.907} C_VEL
LIN {X 0,Y 180.888,Z 293.292,A -85,B 0,C 180,E1 -27886.178,E2 -27886.178} C_VEL
LIN {X 0,Y 179.348,Z 289.089,A -85,B 0,C 180,E1 -27889.13,E2 -27889.13} C_VEL
LIN {X 0,Y 178.37,Z 286.557,A -85,B 0,C 180,E1 -27891.503,E2 -27891.503} C_VEL
LIN {X 0,Y 177.682,Z 284.579,A -85,B 0,C 180,E1 -27893.756,E2 -27893.756} C_VEL
LIN {X 0,Y 176.989,Z 281.431,A -85,B 0,C 180,E1 -27898.863,E2 -27898.863} C_VEL
LIN {X 0,Y 176.991,Z 281.495,A -85,B 0,C 180,E1 -27901.707,E2 -27901.707} C_VEL
LIN {X 0,Y 177.956,Z 285.356,A -85,B 0,C 180,E1 -27907.66,E2 -27907.66} C_VEL
LIN {X 0,Y 179.272,Z 288.975,A -85,B 0,C 180,E1 -27911.161,E2 -27911.161} C_VEL
LIN {X 0,Y 180.732,Z 292.881,A -85,B 0,C 180,E1 -27913.995,E2 -27913.995} C_VEL
LIN {X 0,Y 180.845,Z 293.248,A -85,B 0,C 180,E1 -27914.199,E2 -27914.199} C_VEL
LIN {X 0,Y 177.577,Z 321.104,A -85,B 0,C 180,E1 -27914.866,E2 -27914.866} C_VEL
LIN {X 0,Y 174.449,Z 336.333,A -85,B 0,C 180,E1 -27915.34,E2 -27915.34} C_VEL
LIN {X 0,Y 170.049,Z 351.398,A -85,B 0,C 180,E1 -27916.073,E2 -27916.073} C_VEL
LIN {X 0,Y 164.485,Z 365.887,A -85,B 0,C 180,E1 -27917.054,E2 -27917.054} C_VEL
LIN {X 0,Y 158.198,Z 379.094,A -85,B 0,C 180,E1 -27918.265,E2 -27918.265} C_VEL
LIN {X 0,Y 150.403,Z 392.53,A -85,B 0,C 180,E1 -27919.881,E2 -27919.881} C_VEL
LIN {X 0,Y 141.889,Z 404.729,A -85,B 0,C 180,E1 -27921.764,E2 -27921.764} C_VEL
LIN {X 0,Y 132.855,Z 415.839,A -85,B 0,C 180,E1 -27924.144,E2 -27924.144} C_VEL
LIN {X 0,Y 123.789,Z 425.401,A -85,B 0,C 180,E1 -27926.862,E2 -27926.862} C_VEL
LIN {X 0,Y 114.305,Z 434.354,A -85,B 0,C 180,E1 -27930.595,E2 -27930.595} C_VEL
LIN {X 0,Y 104.899,Z 441.985,A -85,B 0,C 180,E1 -27934.843,E2 -27934.843} C_VEL
LIN {X 0,Y 96.205,Z 448.309,A -85,B 0,C 180,E1 -27939.91,E2 -27939.91} C_VEL
LIN {X 0,Y 88.113,Z 453.646,A -85,B 0,C 180,E1 -27946.124,E2 -27946.124} C_VEL
LIN {X 0,Y 81.721,Z 457.54,A -85,B 0,C 180,E1 -27952.987,E2 -27952.987} C_VEL
LIN {X 0,Y 75.638,Z 461.006,A -85,B 0,C 180,E1 -27962.317,E2 -27962.317} C_VEL
LIN {X 0,Y 71.703,Z 463.283,A -85,B 0,C 180,E1 -27972.9,E2 -27972.9} C_VEL
LIN {X 0,Y 69.918,Z 464.434,A -85,B 0,C 180,E1 -27984.231,E2 -27984.231} C_VEL
LIN {X 0,Y 69.783,Z 464.586,A -85,B 0,C 180,E1 -27990,E2 -27990} C_VEL
LIN {X 0,Y 70.543,Z 464.027,A -85,B 0,C 180,E1 -28001.494,E2 -28001.494} C_VEL
LIN {X 0,Y 73.37,Z 462.357,A -85,B 0,C 180,E1 -28012.529,E2 -28012.529} C_VEL
LIN {X 0,Y 78.355,Z 459.53,A -85,B 0,C 180,E1 -28022.559,E2 -28022.559} C_VEL
LIN {X 0,Y 85.315,Z 455.474,A -85,B 0,C 180,E1 -28031.226,E2 -28031.226} C_VEL
LIN {X 0,Y 93.797,Z 450.089,A -85,B 0,C 180,E1 -28038.529,E2 -28038.529} C_VEL
LIN {X 0,Y 103.544,Z 443.217,A -85,B 0,C 180,E1 -28044.538,E2 -28044.538} C_VEL
LIN {X 0,Y 112.851,Z 435.828,A -85,B 0,C 180,E1 -28048.905,E2 -28048.905} C_VEL
LIN {X 0,Y 122.054,Z 427.383,A -85,B 0,C 180,E1 -28052.571,E2 -28052.571} C_VEL
LIN {X 0,Y 131.289,Z 417.828,A -85,B 0,C 180,E1 -28055.509,E2 -28055.509} C_VEL
LIN {X 0,Y 140.314,Z 407.096,A -85,B 0,C 180,E1 -28057.915,E2 -28057.915} C_VEL
LIN {X 0,Y 148.784,Z 395.373,A -85,B 0,C 180,E1 -28059.856,E2 -28059.856} C_VEL
LIN {X 0,Y 156.4,Z 382.883,A -85,B 0,C 180,E1 -28061.447,E2 -28061.447} C_VEL
LIN {X 0,Y 162.047,Z 371.933,A -85,B 0,C 180,E1 -28062.583,E2 -28062.583} C_VEL
LIN {X 0,Y 168.004,Z 357.96,A -85,B 0,C 180,E1 -28063.645,E2 -28063.645} C_VEL
LIN {X 0,Y 172.814,Z 343.589,A -85,B 0,C 180,E1 -28064.435,E2 -28064.435} C_VEL
LIN {X 0,Y 176.447,Z 328.876,A -85,B 0,C 180,E1 -28065.022,E2 -28065.022} C_VEL
LIN {X 0,Y 178.889,Z 313.76,A -85,B 0,C 180,E1 -28065.44,E2 -28065.44} C_VEL
LIN {X 0,Y 181.125,Z 293.45,A -85,B 0,C 180,E1 -28065.907,E2 -28065.907} C_VEL
LIN {X 0,Y 179.528,Z 289.177,A -85,B 0,C 180,E1 -28068.998,E2 -28068.998} C_VEL
LIN {X 0,Y 178.085,Z 285.006,A -85,B 0,C 180,E1 -28073.058,E2 -28073.058} C_VEL
LIN {X 0,Y 177.299,Z 281.498,A -85,B 0,C 180,E1 -28078.864,E2 -28078.864} C_VEL
LIN {X 0,Y 177.293,Z 281.726,A -85,B 0,C 180,E1 -28081.135,E2 -28081.135} C_VEL
LIN {X 0,Y 178.259,Z 285.553,A -85,B 0,C 180,E1 -28087.219,E2 -28087.219} C_VEL
LIN {X 0,Y 179.635,Z 289.345,A -85,B 0,C 180,E1 -28090.864,E2 -28090.864} C_VEL
LIN {X 0,Y 181.156,Z 293.558,A -85,B 0,C 180,E1 -28093.801,E2 -28093.801} C_VEL
LIN {X 0,Y 177.613,Z 323.715,A -85,B 0,C 180,E1 -28094.497,E2 -28094.497} C_VEL
LIN {X 0,Y 174.559,Z 338.531,A -85,B 0,C 180,E1 -28094.921,E2 -28094.921} C_VEL
LIN {X 0,Y 170.072,Z 353.734,A -85,B 0,C 180,E1 -28095.557,E2 -28095.557} C_VEL
LIN {X 0,Y 164.779,Z 367.446,A -85,B 0,C 180,E1 -28096.33,E2 -28096.33} C_VEL
LIN {X 0,Y 158.323,Z 380.883,A -85,B 0,C 180,E1 -28097.37,E2 -28097.37} C_VEL
LIN {X 0,Y 150.388,Z 394.573,A -85,B 0,C 180,E1 -28098.855,E2 -28098.855} C_VEL
LIN {X 0,Y 141.815,Z 406.978,A -85,B 0,C 180,E1 -28100.707,E2 -28100.707} C_VEL
LIN {X 0,Y 131.829,Z 419.136,A -85,B 0,C 180,E1 -28103.128,E2 -28103.128} C_VEL
LIN {X 0,Y 121.44,Z 429.963,A -85,B 0,C 180,E1 -28106.23,E2 -28106.23} C_VEL
LIN {X 0,Y 111.502,Z 439.005,A -85,B 0,C 180,E1 -28109.95,E2 -28109.95} C_VEL
LIN {X 0,Y 102.289,Z 446.493,A -85,B 0,C 180,E1 -28114.463,E2 -28114.463} C_VEL
LIN {X 0,Y 92.437,Z 453.487,A -85,B 0,C 180,E1 -28120.509,E2 -28120.509} C_VEL
LIN {X 0,Y 83.962,Z 458.999,A -85,B 0,C 180,E1 -28127.96,E2 -28127.96} C_VEL
LIN {X 0,Y 77.117,Z 463.174,A -85,B 0,C 180,E1 -28136.851,E2 -28136.851} C_VEL
LIN {X 0,Y 72.265,Z 466.11,A -85,B 0,C 180,E1 -28147.106,E2 -28147.106} C_VEL
LIN {X 0,Y 69.861,Z 467.874,A -85,B 0,C 180,E1 -28158.393,E2 -28158.393} C_VEL
LIN {X 0,Y 69.666,Z 468.491,A -85,B 0,C 180,E1 -28170,E2 -28170} C_VEL
LIN {X 0,Y 69.858,Z 467.853,A -85,B 0,C 180,E1 -28181.607,E2 -28181.607} C_VEL
LIN {X 0,Y 72.244,Z 466.058,A -85,B 0,C 180,E1 -28192.9,E2 -28192.9} C_VEL
LIN {X 0,Y 77.052,Z 463.096,A -85,B 0,C 180,E1 -28203.18,E2 -28203.18} C_VEL
LIN {X 0,Y 83.888,Z 458.897,A -85,B 0,C 180,E1 -28212.085,E2 -28212.085} C_VEL
LIN {X 0,Y 92.397,Z 453.352,A -85,B 0,C 180,E1 -28219.52,E2 -28219.52} C_VEL
LIN {X 0,Y 102.237,Z 446.315,A -85,B 0,C 180,E1 -28225.579,E2 -28225.579} C_VEL
LIN {X 0,Y 112.875,Z 437.563,A -85,B 0,C 180,E1 -28230.655,E2 -28230.655} C_VEL
LIN {X 0,Y 122.885,Z 428.279,A -85,B 0,C 180,E1 -28234.26,E2 -28234.26} C_VEL
LIN {X 0,Y 131.813,Z 418.85,A -85,B 0,C 180,E1 -28236.888,E2 -28236.888} C_VEL
LIN {X 0,Y 140.127,Z 408.821,A -85,B 0,C 180,E1 -28238.898,E2 -28238.898} C_VEL
LIN {X 0,Y 143.198,Z 404.446,A -85,B 0,C 180,E1 -28239.924,E2 -28239.924} C_VEL
LIN {X 0,Y 147.251,Z 397.196,A -85,B 0,C 180,E1 -28242.074,E2 -28242.074} C_VEL
LIN {X 0,Y 151.125,Z 389.631,A -85,B 0,C 180,E1 -28244.009,E2 -28244.009} C_VEL
LIN {X 0,Y 153.807,Z 384.704,A -85,B 0,C 180,E1 -28244.712,E2 -28244.712} C_VEL
LIN {X 0,Y 160.45,Z 371.946,A -85,B 0,C 180,E1 -28245.724,E2 -28245.724} C_VEL
LIN {X 0,Y 166.225,Z 358.399,A -85,B 0,C 180,E1 -28246.518,E2 -28246.518} C_VEL
LIN {X 0,Y 170.986,Z 344.141,A -85,B 0,C 180,E1 -28247.137,E2 -28247.137} C_VEL
LIN {X 0,Y 174.583,Z 329.369,A -85,B 0,C 180,E1 -28247.619,E2 -28247.619} C_VEL
LIN {X 0,Y 177,Z 313.963,A -85,B 0,C 180,E1 -28247.931,E2 -28247.931} C_VEL
LIN {X 0,Y 178.79,Z 297.749,A -85,B 0,C 180,E1 -28248.302,E2 -28248.302} C_VEL
LIN {X 0,Y 177.479,Z 293.889,A -85,B 0,C 180,E1 -28251.46,E2 -28251.46} C_VEL
LIN {X 0,Y 176.738,Z 291.599,A -85,B 0,C 180,E1 -28253.98,E2 -28253.98} C_VEL
LIN {X 0,Y 176.098,Z 288.421,A -85,B 0,C 180,E1 -28259.429,E2 -28259.429} C_VEL
LIN {X 0,Y 176.108,Z 288.691,A -85,B 0,C 180,E1 -28261.715,E2 -28261.715} C_VEL
LIN {X 0,Y 176.939,Z 292.338,A -85,B 0,C 180,E1 -28267.274,E2 -28267.274} C_VEL
LIN {X 0,Y 178.059,Z 295.716,A -85,B 0,C 180,E1 -28270.527,E2 -28270.527} C_VEL
LIN {X 0,Y 178.775,Z 297.812,A -85,B 0,C 180,E1 -28272.127,E2 -28272.127} C_VEL
LIN {X 0,Y 175.764,Z 321.998,A -85,B 0,C 180,E1 -28272.643,E2 -28272.643} C_VEL
LIN {X 0,Y 172.709,Z 336.542,A -85,B 0,C 180,E1 -28273.072,E2 -28273.072} C_VEL
LIN {X 0,Y 168.224,Z 351.604,A -85,B 0,C 180,E1 -28273.752,E2 -28273.752} C_VEL
LIN {X 0,Y 162.542,Z 366.092,A -85,B 0,C 180,E1 -28274.658,E2 -28274.658} C_VEL
LIN {X 0,Y 155.805,Z 379.859,A -85,B 0,C 180,E1 -28275.849,E2 -28275.849} C_VEL
LIN {X 0,Y 148.14,Z 392.733,A -85,B 0,C 180,E1 -28277.3,E2 -28277.3} C_VEL
LIN {X 0,Y 139.41,Z 404.931,A -85,B 0,C 180,E1 -28279.05,E2 -28279.05} C_VEL
LIN {X 0,Y 130.108,Z 416.041,A -85,B 0,C 180,E1 -28281.285,E2 -28281.285} C_VEL
LIN {X 0,Y 119.542,Z 426.756,A -85,B 0,C 180,E1 -28284.211,E2 -28284.211} C_VEL
LIN {X 0,Y 109.409,Z 435.77,A -85,B 0,C 180,E1 -28287.963,E2 -28287.963} C_VEL
LIN {X 0,Y 99.639,Z 443.186,A -85,B 0,C 180,E1 -28292.176,E2 -28292.176} C_VEL
LIN {X 0,Y 89.29,Z 450.11,A -85,B 0,C 180,E1 -28298.085,E2 -28298.085} C_VEL
LIN {X 0,Y 80.118,Z 455.539,A -85,B 0,C 180,E1 -28305.431,E2 -28305.431} C_VEL
LIN {X 0,Y 72.491,Z 459.627,A -85,B 0,C 180,E1 -28314.43,E2 -28314.43} C_VEL
LIN {X 0,Y 66.905,Z 462.487,A -85,B 0,C 180,E1 -28325.155,E2 -28325.155} C_VEL
LIN {X 0,Y 63.597,Z 464.196,A -85,B 0,C 180,E1 -28337.231,E2 -28337.231} C_VEL
LIN {X 0,Y 62.699,Z 464.784,A -85,B 0,C 180,E1 -28350,E2 -28350} C_VEL
LIN {X 0,Y 63.593,Z 464.225,A -85,B 0,C 180,E1 -28362.77,E2 -28362.77} C_VEL
LIN {X 0,Y 66.827,Z 462.557,A -85,B 0,C 180,E1 -28374.877,E2 -28374.877} C_VEL
LIN {X 0,Y 72.456,Z 459.729,A -85,B 0,C 180,E1 -28385.59,E2 -28385.59} C_VEL
LIN {X 0,Y 80.083,Z 455.673,A -85,B 0,C 180,E1 -28394.594,E2 -28394.594} C_VEL
LIN {X 0,Y 89.237,Z 450.287,A -85,B 0,C 180,E1 -28401.959,E2 -28401.959} C_VEL
LIN {X 0,Y 99.586,Z 443.414,A -85,B 0,C 180,E1 -28407.873,E2 -28407.873} C_VEL
LIN {X 0,Y 109.347,Z 436.025,A -85,B 0,C 180,E1 -28412.098,E2 -28412.098} C_VEL
LIN {X 0,Y 119.479,Z 427.089,A -85,B 0,C 180,E1 -28415.793,E2 -28415.793} C_VEL
LIN {X 0,Y 128.502,Z 418.025,A -85,B 0,C 180,E1 -28418.399,E2 -28418.399} C_VEL
LIN {X 0,Y 137.794,Z 407.292,A -85,B 0,C 180,E1 -28420.66,E2 -28420.66} C_VEL
LIN {X 0,Y 146.492,Z 395.568,A -85,B 0,C 180,E1 -28422.462,E2 -28422.462} C_VEL
LIN {X 0,Y 154.532,Z 382.616,A -85,B 0,C 180,E1 -28424.016,E2 -28424.016} C_VEL
LIN {X 0,Y 160.876,Z 370.379,A -85,B 0,C 180,E1 -28425.141,E2 -28425.141} C_VEL
LIN {X 0,Y 166.968,Z 355.94,A -85,B 0,C 180,E1 -28426.108,E2 -28426.108} C_VEL
LIN {X 0,Y 171.655,Z 341.624,A -85,B 0,C 180,E1 -28426.823,E2 -28426.823} C_VEL
LIN {X 0,Y 175.195,Z 326.89,A -85,B 0,C 180,E1 -28427.334,E2 -28427.334} C_VEL
LIN {X 0,Y 177.553,Z 311.483,A -85,B 0,C 180,E1 -28427.702,E2 -28427.702} C_VEL
LIN {X 0,Y 179.049,Z 297.995,A -85,B 0,C 180,E1 -28428,E2 -28428} C_VEL
LIN {X 0,Y 177.702,Z 294.067,A -85,B 0,C 180,E1 -28431.285,E2 -28431.285} C_VEL
LIN {X 0,Y 176.908,Z 291.591,A -85,B 0,C 180,E1 -28434.133,E2 -28434.133} C_VEL
LIN {X 0,Y 176.418,Z 288.511,A -85,B 0,C 180,E1 -28439.429,E2 -28439.429} C_VEL
LIN {X 0,Y 176.413,Z 288.749,A -85,B 0,C 180,E1 -28440.856,E2 -28440.856} C_VEL
LIN {X 0,Y 177.204,Z 292.414,A -85,B 0,C 180,E1 -28446.69,E2 -28446.69} C_VEL
LIN {X 0,Y 178.362,Z 295.93,A -85,B 0,C 180,E1 -28450.098,E2 -28450.098} C_VEL
LIN {X 0,Y 179.08,Z 298.149,A -85,B 0,C 180,E1 -28451.728,E2 -28451.728} C_VEL
LIN {X 0,Y 176.024,Z 323.224,A -85,B 0,C 180,E1 -28452.249,E2 -28452.249} C_VEL
LIN {X 0,Y 172.866,Z 338.342,A -85,B 0,C 180,E1 -28452.646,E2 -28452.646} C_VEL
LIN {X 0,Y 168.307,Z 353.543,A -85,B 0,C 180,E1 -28453.229,E2 -28453.229} C_VEL
LIN {X 0,Y 162.927,Z 367.254,A -85,B 0,C 180,E1 -28453.937,E2 -28453.937} C_VEL
LIN {X 0,Y 156.344,Z 380.689,A -85,B 0,C 180,E1 -28454.877,E2 -28454.877} C_VEL
LIN {X 0,Y 148.236,Z 394.377,A -85,B 0,C 180,E1 -28456.245,E2 -28456.245} C_VEL
LIN {X 0,Y 139.451,Z 406.781,A -85,B 0,C 180,E1 -28457.962,E2 -28457.962} C_VEL
LIN {X 0,Y 129.199,Z 418.94,A -85,B 0,C 180,E1 -28460.223,E2 -28460.223} C_VEL
LIN {X 0,Y 119.977,Z 428.334,A -85,B 0,C 180,E1 -28462.69,E2 -28462.69} C_VEL
LIN {X 0,Y 109.576,Z 437.577,A -85,B 0,C 180,E1 -28466.111,E2 -28466.111} C_VEL
LIN {X 0,Y 99.739,Z 445.276,A -85,B 0,C 180,E1 -28470.323,E2 -28470.323} C_VEL
LIN {X 0,Y 90.48,Z 451.662,A -85,B 0,C 180,E1 -28475.354,E2 -28475.354} C_VEL
LIN {X 0,Y 80.915,Z 457.54,A -85,B 0,C 180,E1 -28482.414,E2 -28482.414} C_VEL
LIN {X 0,Y 74.775,Z 461.047,A -85,B 0,C 180,E1 -28488.858,E2 -28488.858} C_VEL
LIN {X 0,Y 68.207,Z 464.593,A -85,B 0,C 180,E1 -28498.989,E2 -28498.989} C_VEL
LIN {X 0,Y 63.99,Z 466.937,A -85,B 0,C 180,E1 -28510.762,E2 -28510.762} C_VEL
LIN {X 0,Y 62.447,Z 468.128,A -85,B 0,C 180,E1 -28523.538,E2 -28523.538} C_VEL
LIN {X 0,Y 62.555,Z 468.291,A -85,B 0,C 180,E1 -28530,E2 -28530} C_VEL
LIN {X 0,Y 62.88,Z 467.652,A -85,B 0,C 180,E1 -28542.917,E2 -28542.917} C_VEL
LIN {X 0,Y 65.702,Z 465.857,A -85,B 0,C 180,E1 -28555.332,E2 -28555.332} C_VEL
LIN {X 0,Y 71.159,Z 462.895,A -85,B 0,C 180,E1 -28566.341,E2 -28566.341} C_VEL
LIN {X 0,Y 78.719,Z 458.695,A -85,B 0,C 180,E1 -28575.581,E2 -28575.581} C_VEL
LIN {X 0,Y 87.908,Z 453.15,A -85,B 0,C 180,E1 -28583.08,E2 -28583.08} C_VEL
LIN {X 0,Y 95.686,Z 448.006,A -85,B 0,C 180,E1 -28587.636,E2 -28587.636} C_VEL
LIN {X 0,Y 104.462,Z 441.46,A -85,B 0,C 180,E1 -28591.905,E2 -28591.905} C_VEL
LIN {X 0,Y 113.957,Z 433.613,A -85,B 0,C 180,E1 -28595.46,E2 -28595.46} C_VEL
LIN {X 0,Y 124.531,Z 423.559,A -85,B 0,C 180,E1 -28598.621,E2 -28598.621} C_VEL
LIN {X 0,Y 133.914,Z 413.294,A -85,B 0,C 180,E1 -28600.851,E2 -28600.851} C_VEL
LIN {X 0,Y 143.568,Z 400.86,A -85,B 0,C 180,E1 -28602.86,E2 -28602.86} C_VEL
LIN {X 0,Y 152.275,Z 387.397,A -85,B 0,C 180,E1 -28604.462,E2 -28604.462} C_VEL
LIN {X 0,Y 153.807,Z 384.704,A -85,B 0,C 180,E1 -28604.712,E2 -28604.712} C_VEL
LIN {X 0,Y 156.407,Z 379.732,A -85,B 0,C 180,E1 -28605.369,E2 -28605.369} C_VEL
LIN {X 0,Y 159.839,Z 371.522,A -85,B 0,C 180,E1 -28606.98,E2 -28606.98} C_VEL
LIN {X 0,Y 162.924,Z 363.092,A -85,B 0,C 180,E1 -28608.466,E2 -28608.466} C_VEL
LIN {X 0,Y 164.896,Z 357.705,A -85,B 0,C 180,E1 -28608.942,E2 -28608.942} C_VEL
LIN {X 0,Y 169.755,Z 343.169,A -85,B 0,C 180,E1 -28609.506,E2 -28609.506} C_VEL
LIN {X 0,Y 173.273,Z 328.738,A -85,B 0,C 180,E1 -28609.927,E2 -28609.927} C_VEL
LIN {X 0,Y 175.667,Z 313.628,A -85,B 0,C 180,E1 -28610.196,E2 -28610.196} C_VEL
LIN {X 0,Y 176.924,Z 302.505,A -85,B 0,C 180,E1 -28610.437,E2 -28610.437} C_VEL
LIN {X 0,Y 176.047,Z 299.686,A -85,B 0,C 180,E1 -28613.122,E2 -28613.122} C_VEL
LIN {X 0,Y 175.646,Z 298.279,A -85,B 0,C 180,E1 -28614.835,E2 -28614.835} C_VEL
LIN {X 0,Y 175.23,Z 295.493,A -85,B 0,C 180,E1 -28619.426,E2 -28619.426} C_VEL
LIN {X 0,Y 175.226,Z 295.705,A -85,B 0,C 180,E1 -28621.437,E2 -28621.437} C_VEL
LIN {X 0,Y 175.866,Z 299.04,A -85,B 0,C 180,E1 -28626.598,E2 -28626.598} C_VEL
LIN {X 0,Y 176.893,Z 302.479,A -85,B 0,C 180,E1 -28629.938,E2 -28629.938} C_VEL
LIN {X 0,Y 174.165,Z 323.186,A -85,B 0,C 180,E1 -28630.381,E2 -28630.381} C_VEL
LIN {X 0,Y 170.979,Z 337.733,A -85,B 0,C 180,E1 -28630.803,E2 -28630.803} C_VEL
LIN {X 0,Y 166.645,Z 351.905,A -85,B 0,C 180,E1 -28631.389,E2 -28631.389} C_VEL
LIN {X 0,Y 160.896,Z 366.296,A -85,B 0,C 180,E1 -28632.218,E2 -28632.218} C_VEL
LIN {X 0,Y 154.012,Z 380.063,A -85,B 0,C 180,E1 -28633.298,E2 -28633.298} C_VEL
LIN {X 0,Y 146.186,Z 392.935,A -85,B 0,C 180,E1 -28634.641,E2 -28634.641} C_VEL
LIN {X 0,Y 137.261,Z 405.133,A -85,B 0,C 180,E1 -28636.253,E2 -28636.253} C_VEL
LIN {X 0,Y 127.698,Z 416.243,A -85,B 0,C 180,E1 -28638.309,E2 -28638.309} C_VEL
LIN {X 0,Y 116.489,Z 427.23,A -85,B 0,C 180,E1 -28641.109,E2 -28641.109} C_VEL
LIN {X 0,Y 106.262,Z 435.971,A -85,B 0,C 180,E1 -28644.576,E2 -28644.576} C_VEL
LIN {X 0,Y 96.04,Z 443.387,A -85,B 0,C 180,E1 -28648.582,E2 -28648.582} C_VEL
LIN {X 0,Y 85.082,Z 450.31,A -85,B 0,C 180,E1 -28654.307,E2 -28654.307} C_VEL
LIN {X 0,Y 75.201,Z 455.74,A -85,B 0,C 180,E1 -28661.613,E2 -28661.613} C_VEL
LIN {X 0,Y 66.83,Z 459.827,A -85,B 0,C 180,E1 -28670.878,E2 -28670.878} C_VEL
LIN {X 0,Y 60.496,Z 462.688,A -85,B 0,C 180,E1 -28682.31,E2 -28682.31} C_VEL
LIN {X 0,Y 56.681,Z 464.396,A -85,B 0,C 180,E1 -28695.642,E2 -28695.642} C_VEL
LIN {X 0,Y 55.608,Z 464.983,A -85,B 0,C 180,E1 -28710,E2 -28710} C_VEL
LIN {X 0,Y 56.674,Z 464.424,A -85,B 0,C 180,E1 -28724.36,E2 -28724.36} C_VEL
LIN {X 0,Y 60.425,Z 462.756,A -85,B 0,C 180,E1 -28737.726,E2 -28737.726} C_VEL
LIN {X 0,Y 66.799,Z 459.928,A -85,B 0,C 180,E1 -28749.144,E2 -28749.144} C_VEL
LIN {X 0,Y 75.166,Z 455.871,A -85,B 0,C 180,E1 -28758.418,E2 -28758.418} C_VEL
LIN {X 0,Y 85.026,Z 450.485,A -85,B 0,C 180,E1 -28765.748,E2 -28765.748} C_VEL
LIN {X 0,Y 95.978,Z 443.613,A -85,B 0,C 180,E1 -28771.487,E2 -28771.487} C_VEL
LIN {X 0,Y 106.204,Z 436.222,A -85,B 0,C 180,E1 -28775.492,E2 -28775.492} C_VEL
LIN {X 0,Y 116.437,Z 427.553,A -85,B 0,C 180,E1 -28778.893,E2 -28778.893} C_VEL
LIN {X 0,Y 126.061,Z 418.221,A -85,B 0,C 180,E1 -28781.4,E2 -28781.4} C_VEL
LIN {X 0,Y 135.607,Z 407.488,A -85,B 0,C 180,E1 -28783.494,E2 -28783.494} C_VEL
LIN {X 0,Y 144.512,Z 395.763,A -85,B 0,C 180,E1 -28785.146,E2 -28785.146} C_VEL
LIN {X 0,Y 152.723,Z 382.811,A -85,B 0,C 180,E1 -28786.588,E2 -28786.588} C_VEL
LIN {X 0,Y 159.202,Z 370.572,A -85,B 0,C 180,E1 -28787.613,E2 -28787.613} C_VEL
LIN {X 0,Y 165.409,Z 356.131,A -85,B 0,C 180,E1 -28788.492,E2 -28788.492} C_VEL
LIN {X 0,Y 170.181,Z 341.813,A -85,B 0,C 180,E1 -28789.145,E2 -28789.145} C_VEL
LIN {X 0,Y 173.659,Z 327.723,A -85,B 0,C 180,E1 -28789.596,E2 -28789.596} C_VEL
LIN {X 0,Y 176.161,Z 311.811,A -85,B 0,C 180,E1 -28789.953,E2 -28789.953} C_VEL
LIN {X 0,Y 177.179,Z 302.711,A -85,B 0,C 180,E1 -28790.172,E2 -28790.172} C_VEL
LIN {X 0,Y 176.036,Z 298.726,A -85,B 0,C 180,E1 -28794.104,E2 -28794.104} C_VEL
LIN {X 0,Y 175.555,Z 295.539,A -85,B 0,C 180,E1 -28799.426,E2 -28799.426} C_VEL
LIN {X 0,Y 175.527,Z 296.033,A -85,B 0,C 180,E1 -28801.003,E2 -28801.003} C_VEL
LIN {X 0,Y 176.202,Z 299.374,A -85,B 0,C 180,E1 -28806.297,E2 -28806.297} C_VEL
LIN {X 0,Y 177.2,Z 302.738,A -85,B 0,C 180,E1 -28809.526,E2 -28809.526} C_VEL
LIN {X 0,Y 174.457,Z 324.133,A -85,B 0,C 180,E1 -28810.002,E2 -28810.002} C_VEL
LIN {X 0,Y 171.197,Z 339.082,A -85,B 0,C 180,E1 -28810.361,E2 -28810.361} C_VEL
LIN {X 0,Y 166.827,Z 353.351,A -85,B 0,C 180,E1 -28810.856,E2 -28810.856} C_VEL
LIN {X 0,Y 161.363,Z 367.061,A -85,B 0,C 180,E1 -28811.487,E2 -28811.487} C_VEL
LIN {X 0,Y 154.671,Z 380.494,A -85,B 0,C 180,E1 -28812.331,E2 -28812.331} C_VEL
LIN {X 0,Y 146.407,Z 394.182,A -85,B 0,C 180,E1 -28813.572,E2 -28813.572} C_VEL
LIN {X 0,Y 137.41,Z 406.584,A -85,B 0,C 180,E1 -28815.118,E2 -28815.118} C_VEL
LIN {X 0,Y 126.915,Z 418.743,A -85,B 0,C 180,E1 -28817.208,E2 -28817.208} C_VEL
LIN {X 0,Y 117.402,Z 428.136,A -85,B 0,C 180,E1 -28819.466,E2 -28819.466} C_VEL
LIN {X 0,Y 106.608,Z 437.378,A -85,B 0,C 180,E1 -28822.641,E2 -28822.641} C_VEL
LIN {X 0,Y 96.323,Z 445.077,A -85,B 0,C 180,E1 -28826.645,E2 -28826.645} C_VEL
LIN {X 0,Y 86.529,Z 451.463,A -85,B 0,C 180,E1 -28831.479,E2 -28831.479} C_VEL
LIN {X 0,Y 76.266,Z 457.341,A -85,B 0,C 180,E1 -28838.437,E2 -28838.437} C_VEL
LIN {X 0,Y 69.203,Z 461.007,A -85,B 0,C 180,E1 -28845.306,E2 -28845.306} C_VEL
LIN {X 0,Y 62.173,Z 464.393,A -85,B 0,C 180,E1 -28855.583,E2 -28855.583} C_VEL
LIN {X 0,Y 57.278,Z 466.737,A -85,B 0,C 180,E1 -28868.401,E2 -28868.401} C_VEL
LIN {X 0,Y 55.366,Z 467.928,A -85,B 0,C 180,E1 -28882.707,E2 -28882.707} C_VEL
LIN {X 0,Y 55.463,Z 468.093,A -85,B 0,C 180,E1 -28890,E2 -28890} C_VEL
LIN {X 0,Y 55.953,Z 467.453,A -85,B 0,C 180,E1 -28904.549,E2 -28904.549} C_VEL
LIN {X 0,Y 59.312,Z 465.656,A -85,B 0,C 180,E1 -28918.292,E2 -28918.292} C_VEL
LIN {X 0,Y 65.521,Z 462.693,A -85,B 0,C 180,E1 -28930.059,E2 -28930.059} C_VEL
LIN {X 0,Y 73.868,Z 458.493,A -85,B 0,C 180,E1 -28939.565,E2 -28939.565} C_VEL
LIN {X 0,Y 83.798,Z 452.948,A -85,B 0,C 180,E1 -28947.001,E2 -28947.001} C_VEL
LIN {X 0,Y 94.844,Z 445.908,A -85,B 0,C 180,E1 -28952.774,E2 -28952.774} C_VEL
LIN {X 0,Y 105.076,Z 438.385,A -85,B 0,C 180,E1 -28956.878,E2 -28956.878} C_VEL
LIN {X 0,Y 115.826,Z 429.329,A -85,B 0,C 180,E1 -28960.135,E2 -28960.135} C_VEL
LIN {X 0,Y 125.291,Z 420.087,A -85,B 0,C 180,E1 -28962.477,E2 -28962.477} C_VEL
LIN {X 0,Y 134.987,Z 409.207,A -85,B 0,C 180,E1 -28964.406,E2 -28964.406} C_VEL
LIN {X 0,Y 143.594,Z 397.812,A -85,B 0,C 180,E1 -28965.984,E2 -28965.984} C_VEL
LIN {X 0,Y 151.773,Z 385.032,A -85,B 0,C 180,E1 -28967.26,E2 -28967.26} C_VEL
LIN {X 0,Y 158.841,Z 371.741,A -85,B 0,C 180,E1 -28968.219,E2 -28968.219} C_VEL
LIN {X 0,Y 164.896,Z 357.705,A -85,B 0,C 180,E1 -28968.942,E2 -28968.942} C_VEL
LIN {X 0,Y 166.797,Z 352.235,A -85,B 0,C 180,E1 -28969.379,E2 -28969.379} C_VEL
LIN {X 0,Y 170.663,Z 336.159,A -85,B 0,C 180,E1 -28971.686,E2 -28971.686} C_VEL
LIN {X 0,Y 171.786,Z 330.535,A -85,B 0,C 180,E1 -28972.174,E2 -28972.174} C_VEL
LIN {X 0,Y 172.16,Z 328.611,A -85,B 0,C 180,E1 -28972.246,E2 -28972.246} C_VEL
LIN {X 0,Y 174.597,Z 313.406,A -85,B 0,C 180,E1 -28972.496,E2 -28972.496} C_VEL
LIN {X 0,Y 175.273,Z 307.421,A -85,B 0,C 180,E1 -28972.657,E2 -28972.657} C_VEL
LIN {X 0,Y 174.654,Z 305.105,A -85,B 0,C 180,E1 -28975.384,E2 -28975.384} C_VEL
LIN {X 0,Y 174.361,Z 302.569,A -85,B 0,C 180,E1 -28979.424,E2 -28979.424} C_VEL
LIN {X 0,Y 174.342,Z 302.781,A -85,B 0,C 180,E1 -28981.178,E2 -28981.178} C_VEL
LIN {X 0,Y 174.842,Z 305.899,A -85,B 0,C 180,E1 -28986.057,E2 -28986.057} C_VEL
LIN {X 0,Y 175.258,Z 307.459,A -85,B 0,C 180,E1 -28987.758,E2 -28987.758} C_VEL
LIN {X 0,Y 172.844,Z 324.409,A -85,B 0,C 180,E1 -28988.1,E2 -28988.1} C_VEL
LIN {X 0,Y 169.644,Z 338.479,A -85,B 0,C 180,E1 -28988.469,E2 -28988.469} C_VEL
LIN {X 0,Y 164.88,Z 353.487,A -85,B 0,C 180,E1 -28989.051,E2 -28989.051} C_VEL
LIN {X 0,Y 159.547,Z 366.5,A -85,B 0,C 180,E1 -28989.73,E2 -28989.73} C_VEL
LIN {X 0,Y 152.533,Z 380.267,A -85,B 0,C 180,E1 -28990.697,E2 -28990.697} C_VEL
LIN {X 0,Y 144.55,Z 393.138,A -85,B 0,C 180,E1 -28991.909,E2 -28991.909} C_VEL
LIN {X 0,Y 135.447,Z 405.334,A -85,B 0,C 180,E1 -28993.372,E2 -28993.372} C_VEL
LIN {X 0,Y 125.648,Z 416.445,A -85,B 0,C 180,E1 -28995.233,E2 -28995.233} C_VEL
LIN {X 0,Y 114.352,Z 427.233,A -85,B 0,C 180,E1 -28997.713,E2 -28997.713} C_VEL
LIN {X 0,Y 103.504,Z 436.172,A -85,B 0,C 180,E1 -29000.991,E2 -29000.991} C_VEL
LIN {X 0,Y 92.835,Z 443.589,A -85,B 0,C 180,E1 -29004.707,E2 -29004.707} C_VEL
LIN {X 0,Y 81.277,Z 450.511,A -85,B 0,C 180,E1 -29010.151,E2 -29010.151} C_VEL
LIN {X 0,Y 70.668,Z 455.941,A -85,B 0,C 180,E1 -29017.287,E2 -29017.287} C_VEL
LIN {X 0,Y 61.475,Z 460.027,A -85,B 0,C 180,E1 -29026.691,E2 -29026.691} C_VEL
LIN {X 0,Y 54.277,Z 462.888,A -85,B 0,C 180,E1 -29038.807,E2 -29038.807} C_VEL
LIN {X 0,Y 49.832,Z 464.595,A -85,B 0,C 180,E1 -29053.617,E2 -29053.617} C_VEL
LIN {X 0,Y 48.508,Z 465.182,A -85,B 0,C 180,E1 -29070,E2 -29070} C_VEL
LIN {X 0,Y 49.824,Z 464.623,A -85,B 0,C 180,E1 -29086.387,E2 -29086.387} C_VEL
LIN {X 0,Y 54.215,Z 462.955,A -85,B 0,C 180,E1 -29101.234,E2 -29101.234} C_VEL
LIN {X 0,Y 61.445,Z 460.126,A -85,B 0,C 180,E1 -29113.336,E2 -29113.336} C_VEL
LIN {X 0,Y 70.634,Z 456.07,A -85,B 0,C 180,E1 -29122.75,E2 -29122.75} C_VEL
LIN {X 0,Y 81.222,Z 450.684,A -85,B 0,C 180,E1 -29129.916,E2 -29129.916} C_VEL
LIN {X 0,Y 92.781,Z 443.811,A -85,B 0,C 180,E1 -29135.365,E2 -29135.365} C_VEL
LIN {X 0,Y 103.454,Z 436.42,A -85,B 0,C 180,E1 -29139.082,E2 -29139.082} C_VEL
LIN {X 0,Y 114.023,Z 427.783,A -85,B 0,C 180,E1 -29142.231,E2 -29142.231} C_VEL
LIN {X 0,Y 123.982,Z 418.417,A -85,B 0,C 180,E1 -29144.506,E2 -29144.506} C_VEL
LIN {X 0,Y 133.764,Z 407.684,A -85,B 0,C 180,E1 -29146.409,E2 -29146.409} C_VEL
LIN {X 0,Y 142.857,Z 395.958,A -85,B 0,C 180,E1 -29147.898,E2 -29147.898} C_VEL
LIN {X 0,Y 151.222,Z 383.021,A -85,B 0,C 180,E1 -29149.21,E2 -29149.21} C_VEL
LIN {X 0,Y 158.674,Z 369.003,A -85,B 0,C 180,E1 -29150.232,E2 -29150.232} C_VEL
LIN {X 0,Y 164.918,Z 354.259,A -85,B 0,C 180,E1 -29151,E2 -29151} C_VEL
LIN {X 0,Y 169.78,Z 339.148,A -85,B 0,C 180,E1 -29151.601,E2 -29151.601} C_VEL
LIN {X 0,Y 173.315,Z 323.615,A -85,B 0,C 180,E1 -29152.014,E2 -29152.014} C_VEL
LIN {X 0,Y 175.55,Z 307.723,A -85,B 0,C 180,E1 -29152.341,E2 -29152.341} C_VEL
LIN {X 0,Y 174.942,Z 305.332,A -85,B 0,C 180,E1 -29155.103,E2 -29155.103} C_VEL
LIN {X 0,Y 174.684,Z 302.599,A -85,B 0,C 180,E1 -29160,E2 -29160} C_VEL
LIN {X 0,Y 175.181,Z 306.187,A -85,B 0,C 180,E1 -29165.756,E2 -29165.756} C_VEL
LIN {X 0,Y 175.565,Z 307.673,A -85,B 0,C 180,E1 -29167.331,E2 -29167.331} C_VEL
LIN {X 0,Y 173.951,Z 320.43,A -85,B 0,C 180,E1 -29167.605,E2 -29167.605} C_VEL
LIN {X 0,Y 170.793,Z 336.09,A -85,B 0,C 180,E1 -29167.935,E2 -29167.935} C_VEL
LIN {X 0,Y 166.379,Z 351.032,A -85,B 0,C 180,E1 -29168.38,E2 -29168.38} C_VEL
LIN {X 0,Y 160.948,Z 364.89,A -85,B 0,C 180,E1 -29168.902,E2 -29168.902} C_VEL
LIN {X 0,Y 154.157,Z 378.716,A -85,B 0,C 180,E1 -29169.637,E2 -29169.637} C_VEL
LIN {X 0,Y 146.573,Z 391.4,A -85,B 0,C 180,E1 -29170.593,E2 -29170.593} C_VEL
LIN {X 0,Y 137.762,Z 403.765,A -85,B 0,C 180,E1 -29171.895,E2 -29171.895} C_VEL
LIN {X 0,Y 128.286,Z 414.999,A -85,B 0,C 180,E1 -29173.488,E2 -29173.488} C_VEL
LIN {X 0,Y 118.448,Z 424.953,A -85,B 0,C 180,E1 -29175.381,E2 -29175.381} C_VEL
LIN {X 0,Y 107.209,Z 434.701,A -85,B 0,C 180,E1 -29178.095,E2 -29178.095} C_VEL
LIN {X 0,Y 97.194,Z 442.241,A -85,B 0,C 180,E1 -29181.195,E2 -29181.195} C_VEL
LIN {X 0,Y 85.919,Z 449.591,A -85,B 0,C 180,E1 -29185.87,E2 -29185.87} C_VEL
LIN {X 0,Y 74.663,Z 455.818,A -85,B 0,C 180,E1 -29192.094,E2 -29192.094} C_VEL
LIN {X 0,Y 63.678,Z 461.101,A -85,B 0,C 180,E1 -29201.467,E2 -29201.467} C_VEL
LIN {X 0,Y 56.398,Z 464.193,A -85,B 0,C 180,E1 -29211.459,E2 -29211.459} C_VEL
LIN {X 0,Y 50.679,Z 466.536,A -85,B 0,C 180,E1 -29225.415,E2 -29225.415} C_VEL
LIN {X 0,Y 48.316,Z 467.729,A -85,B 0,C 180,E1 -29241.636,E2 -29241.636} C_VEL
LIN {X 0,Y 48.355,Z 467.894,A -85,B 0,C 180,E1 -29250,E2 -29250} C_VEL
LIN {X 0,Y 49.063,Z 467.252,A -85,B 0,C 180,E1 -29266.648,E2 -29266.648} C_VEL
LIN {X 0,Y 53.123,Z 465.456,A -85,B 0,C 180,E1 -29281.95,E2 -29281.95} C_VEL
LIN {X 0,Y 60.196,Z 462.491,A -85,B 0,C 180,E1 -29294.468,E2 -29294.468} C_VEL
LIN {X 0,Y 69.441,Z 458.292,A -85,B 0,C 180,E1 -29304.063,E2 -29304.063} C_VEL
LIN {X 0,Y 80.12,Z 452.746,A -85,B 0,C 180,E1 -29311.304,E2 -29311.304} C_VEL
LIN {X 0,Y 91.789,Z 445.706,A -85,B 0,C 180,E1 -29316.751,E2 -29316.751} C_VEL
LIN {X 0,Y 102.479,Z 438.183,A -85,B 0,C 180,E1 -29320.557,E2 -29320.557} C_VEL
LIN {X 0,Y 113.594,Z 429.126,A -85,B 0,C 180,E1 -29323.532,E2 -29323.532} C_VEL
LIN {X 0,Y 123.336,Z 419.885,A -85,B 0,C 180,E1 -29325.629,E2 -29325.629} C_VEL
LIN {X 0,Y 133.243,Z 409.004,A -85,B 0,C 180,E1 -29327.369,E2 -29327.369} C_VEL
LIN {X 0,Y 141.888,Z 397.812,A -85,B 0,C 180,E1 -29328.76,E2 -29328.76} C_VEL
LIN {X 0,Y 149.934,Z 385.559,A -85,B 0,C 180,E1 -29329.853,E2 -29329.853} C_VEL
LIN {X 0,Y 157.539,Z 371.535,A -85,B 0,C 180,E1 -29330.759,E2 -29330.759} C_VEL
LIN {X 0,Y 163.891,Z 356.946,A -85,B 0,C 180,E1 -29331.403,E2 -29331.403} C_VEL
LIN {X 0,Y 168.897,Z 341.924,A -85,B 0,C 180,E1 -29331.904,E2 -29331.904} C_VEL
LIN {X 0,Y 172.16,Z 328.611,A -85,B 0,C 180,E1 -29332.246,E2 -29332.246} C_VEL
LIN {X 0,Y 172.875,Z 324.44,A -85,B 0,C 180,E1 -29332.511,E2 -29332.511} C_VEL
LIN {X 0,Y 173.346,Z 320.49,A -85,B 0,C 180,E1 -29333.068,E2 -29333.068} C_VEL
LIN {X 0,Y 173.643,Z 315.889,A -85,B 0,C 180,E1 -29334.165,E2 -29334.165} C_VEL
LIN {X 0,Y 173.695,Z 313.232,A -85,B 0,C 180,E1 -29335.234,E2 -29335.234} C_VEL
LIN {X 0,Y 173.594,Z 311.664,A -85,B 0,C 180,E1 -29336.497,E2 -29336.497} C_VEL
LIN {X 0,Y 173.492,Z 309.515,A -85,B 0,C 180,E1 -29340,E2 -29340} C_VEL
LIN {X 0,Y 173.459,Z 310.731,A -85,B 0,C 180,E1 -29342.322,E2 -29342.322} C_VEL
LIN {X 0,Y 173.838,Z 312.776,A -85,B 0,C 180,E1 -29345.532,E2 -29345.532} C_VEL
LIN {X 0,Y 171.308,Z 328.234,A -85,B 0,C 180,E1 -29345.834,E2 -29345.834} C_VEL
LIN {X 0,Y 168.294,Z 340.299,A -85,B 0,C 180,E1 -29346.141,E2 -29346.141} C_VEL
LIN {X 0,Y 163.457,Z 354.901,A -85,B 0,C 180,E1 -29346.658,E2 -29346.658} C_VEL
LIN {X 0,Y 157.65,Z 368.465,A -85,B 0,C 180,E1 -29347.297,E2 -29347.297} C_VEL
LIN {X 0,Y 150.232,Z 382.398,A -85,B 0,C 180,E1 -29348.216,E2 -29348.216} C_VEL
LIN {X 0,Y 141.568,Z 395.678,A -85,B 0,C 180,E1 -29349.363,E2 -29349.363} C_VEL
LIN {X 0,Y 132.302,Z 407.48,A -85,B 0,C 180,E1 -29350.66,E2 -29350.66} C_VEL
LIN {X 0,Y 122.304,Z 418.275,A -85,B 0,C 180,E1 -29352.344,E2 -29352.344} C_VEL
LIN {X 0,Y 112.395,Z 427.434,A -85,B 0,C 180,E1 -29354.263,E2 -29354.263} C_VEL
LIN {X 0,Y 101.17,Z 436.373,A -85,B 0,C 180,E1 -29357.221,E2 -29357.221} C_VEL
LIN {X 0,Y 90.083,Z 443.79,A -85,B 0,C 180,E1 -29360.577,E2 -29360.577} C_VEL
LIN {X 0,Y 77.936,Z 450.712,A -85,B 0,C 180,E1 -29365.609,E2 -29365.609} C_VEL
LIN {X 0,Y 66.59,Z 456.141,A -85,B 0,C 180,E1 -29372.399,E2 -29372.399} C_VEL
LIN {X 0,Y 56.489,Z 460.228,A -85,B 0,C 180,E1 -29381.714,E2 -29381.714} C_VEL
LIN {X 0,Y 48.321,Z 463.088,A -85,B 0,C 180,E1 -29394.424,E2 -29394.424} C_VEL
LIN {X 0,Y 43.05,Z 464.794,A -85,B 0,C 180,E1 -29410.943,E2 -29410.943} C_VEL
LIN {X 0,Y 41.426,Z 465.38,A -85,B 0,C 180,E1 -29430,E2 -29430} C_VEL
LIN {X 0,Y 43.04,Z 464.822,A -85,B 0,C 180,E1 -29449.062,E2 -29449.062} C_VEL
LIN {X 0,Y 48.267,Z 463.154,A -85,B 0,C 180,E1 -29465.622,E2 -29465.622} C_VEL
LIN {X 0,Y 56.46,Z 460.325,A -85,B 0,C 180,E1 -29478.32,E2 -29478.32} C_VEL
LIN {X 0,Y 66.56,Z 456.269,A -85,B 0,C 180,E1 -29487.641,E2 -29487.641} C_VEL
LIN {X 0,Y 77.897,Z 450.882,A -85,B 0,C 180,E1 -29494.452,E2 -29494.452} C_VEL
LIN {X 0,Y 90.035,Z 444.01,A -85,B 0,C 180,E1 -29499.506,E2 -29499.506} C_VEL
LIN {X 0,Y 102.723,Z 435.422,A -85,B 0,C 180,E1 -29503.304,E2 -29503.304} C_VEL
LIN {X 0,Y 113.848,Z 426.445,A -85,B 0,C 180,E1 -29506.104,E2 -29506.104} C_VEL
LIN {X 0,Y 123.943,Z 416.993,A -85,B 0,C 180,E1 -29507.998,E2 -29507.998} C_VEL
LIN {X 0,Y 134.789,Z 404.94,A -85,B 0,C 180,E1 -29509.788,E2 -29509.788} C_VEL
LIN {X 0,Y 144.075,Z 392.624,A -85,B 0,C 180,E1 -29511.044,E2 -29511.044} C_VEL
LIN {X 0,Y 152.175,Z 379.644,A -85,B 0,C 180,E1 -29512.157,E2 -29512.157} C_VEL
LIN {X 0,Y 159.335,Z 365.657,A -85,B 0,C 180,E1 -29512.952,E2 -29512.952} C_VEL
LIN {X 0,Y 165.306,Z 350.863,A -85,B 0,C 180,E1 -29513.585,E2 -29513.585} C_VEL
LIN {X 0,Y 169.953,Z 335.463,A -85,B 0,C 180,E1 -29514.086,E2 -29514.086} C_VEL
LIN {X 0,Y 173.172,Z 319.931,A -85,B 0,C 180,E1 -29514.403,E2 -29514.403} C_VEL
LIN {X 0,Y 174.134,Z 313.027,A -85,B 0,C 180,E1 -29514.572,E2 -29514.572} C_VEL
LIN {X 0,Y 173.782,Z 309.98,A -85,B 0,C 180,E1 -29519.42,E2 -29519.42} C_VEL
LIN {X 0,Y 173.784,Z 309.975,A -85,B 0,C 180,E1 -29520.289,E2 -29520.289} C_VEL
LIN {X 0,Y 174.163,Z 312.961,A -85,B 0,C 180,E1 -29525.152,E2 -29525.152} C_VEL
LIN {X 0,Y 171.505,Z 329.302,A -85,B 0,C 180,E1 -29525.435,E2 -29525.435} C_VEL
LIN {X 0,Y 167.49,Z 344.786,A -85,B 0,C 180,E1 -29525.768,E2 -29525.768} C_VEL
LIN {X 0,Y 162.158,Z 359.716,A -85,B 0,C 180,E1 -29526.213,E2 -29526.213} C_VEL
LIN {X 0,Y 155.704,Z 373.755,A -85,B 0,C 180,E1 -29526.773,E2 -29526.773} C_VEL
LIN {X 0,Y 147.996,Z 387.304,A -85,B 0,C 180,E1 -29527.557,E2 -29527.557} C_VEL
LIN {X 0,Y 139.467,Z 399.722,A -85,B 0,C 180,E1 -29528.575,E2 -29528.575} C_VEL
LIN {X 0,Y 130.188,Z 411.117,A -85,B 0,C 180,E1 -29529.868,E2 -29529.868} C_VEL
LIN {X 0,Y 120.089,Z 421.615,A -85,B 0,C 180,E1 -29531.4,E2 -29531.4} C_VEL
LIN {X 0,Y 108.491,Z 431.893,A -85,B 0,C 180,E1 -29533.663,E2 -29533.663} C_VEL
LIN {X 0,Y 97.117,Z 440.443,A -85,B 0,C 180,E1 -29536.492,E2 -29536.492} C_VEL
LIN {X 0,Y 86.121,Z 447.568,A -85,B 0,C 180,E1 -29540.203,E2 -29540.203} C_VEL
LIN {X 0,Y 74.003,Z 454.18,A -85,B 0,C 180,E1 -29545.549,E2 -29545.549} C_VEL
LIN {X 0,Y 62.844,Z 459.365,A -85,B 0,C 180,E1 -29552.991,E2 -29552.991} C_VEL
LIN {X 0,Y 55.369,Z 462.374,A -85,B 0,C 180,E1 -29560.396,E2 -29560.396} C_VEL
LIN {X 0,Y 47.232,Z 465.31,A -85,B 0,C 180,E1 -29573.473,E2 -29573.473} C_VEL
LIN {X 0,Y 42.273,Z 467.075,A -85,B 0,C 180,E1 -29590.579,E2 -29590.579} C_VEL
LIN {X 0,Y 41.264,Z 467.695,A -85,B 0,C 180,E1 -29610,E2 -29610} C_VEL
LIN {X 0,Y 42.269,Z 467.052,A -85,B 0,C 180,E1 -29629.423,E2 -29629.423} C_VEL
LIN {X 0,Y 47.209,Z 465.255,A -85,B 0,C 180,E1 -29646.547,E2 -29646.547} C_VEL
LIN {X 0,Y 55.301,Z 462.29,A -85,B 0,C 180,E1 -29659.686,E2 -29659.686} C_VEL
LIN {X 0,Y 65.491,Z 458.09,A -85,B 0,C 180,E1 -29669.148,E2 -29669.148} C_VEL
LIN {X 0,Y 76.937,Z 452.544,A -85,B 0,C 180,E1 -29675.991,E2 -29675.991} C_VEL
LIN {X 0,Y 89.203,Z 445.504,A -85,B 0,C 180,E1 -29680.987,E2 -29680.987} C_VEL
LIN {X 0,Y 100.326,Z 437.981,A -85,B 0,C 180,E1 -29684.41,E2 -29684.41} C_VEL
LIN {X 0,Y 111.776,Z 428.924,A -85,B 0,C 180,E1 -29687.053,E2 -29687.053} C_VEL
LIN {X 0,Y 121.76,Z 419.683,A -85,B 0,C 180,E1 -29688.885,E2 -29688.885} C_VEL
LIN {X 0,Y 131.863,Z 408.801,A -85,B 0,C 180,E1 -29690.405,E2 -29690.405} C_VEL
LIN {X 0,Y 141.266,Z 396.793,A -85,B 0,C 180,E1 -29691.671,E2 -29691.671} C_VEL
LIN {X 0,Y 149.702,Z 383.925,A -85,B 0,C 180,E1 -29692.636,E2 -29692.636} C_VEL
LIN {X 0,Y 157.415,Z 369.562,A -85,B 0,C 180,E1 -29693.405,E2 -29693.405} C_VEL
LIN {X 0,Y 163.294,Z 355.915,A -85,B 0,C 180,E1 -29693.903,E2 -29693.903} C_VEL
LIN {X 0,Y 168.248,Z 341.006,A -85,B 0,C 180,E1 -29694.308,E2 -29694.308} C_VEL
LIN {X 0,Y 171.919,Z 325.393,A -85,B 0,C 180,E1 -29694.63,E2 -29694.63} C_VEL
LIN {X 0,Y 173.861,Z 312.747,A -85,B 0,C 180,E1 -29694.837,E2 -29694.837} C_VEL
LIN {X 0,Y 173.594,Z 311.664,A -85,B 0,C 180,E1 -29696.497,E2 -29696.497} C_VEL
LIN {X 0,Y 173.387,Z 311.671,A -85,B 0,C 180,E1 -29697.78,E2 -29697.78} C_VEL
LIN {X 0,Y 173.129,Z 312.795,A -85,B 0,C 180,E1 -29699.035,E2 -29699.035} C_VEL
LIN {X 0,Y 172.509,Z 318.009,A -85,B 0,C 180,E1 -29702.742,E2 -29702.742} C_VEL
LIN {X 0,Y 172.518,Z 318.373,A -85,B 0,C 180,E1 -29703.184,E2 -29703.184} C_VEL
LIN {X 0,Y 172.528,Z 318.417,A -85,B 0,C 180,E1 -29703.294,E2 -29703.294} C_VEL
LIN {X 0,Y 169.427,Z 333.982,A -85,B 0,C 180,E1 -29703.548,E2 -29703.548} C_VEL
LIN {X 0,Y 165.19,Z 348.486,A -85,B 0,C 180,E1 -29703.972,E2 -29703.972} C_VEL
LIN {X 0,Y 160.359,Z 361.097,A -85,B 0,C 180,E1 -29704.395,E2 -29704.395} C_VEL
LIN {X 0,Y 153.657,Z 375.066,A -85,B 0,C 180,E1 -29705.065,E2 -29705.065} C_VEL
LIN {X 0,Y 146.595,Z 387.158,A -85,B 0,C 180,E1 -29705.852,E2 -29705.852} C_VEL
LIN {X 0,Y 138.017,Z 399.375,A -85,B 0,C 180,E1 -29706.8,E2 -29706.8} C_VEL
LIN {X 0,Y 127.772,Z 411.537,A -85,B 0,C 180,E1 -29708.076,E2 -29708.076} C_VEL
LIN {X 0,Y 117.6,Z 421.716,A -85,B 0,C 180,E1 -29709.574,E2 -29709.574} C_VEL
LIN {X 0,Y 105.84,Z 431.675,A -85,B 0,C 180,E1 -29711.666,E2 -29711.666} C_VEL
LIN {X 0,Y 95.994,Z 438.798,A -85,B 0,C 180,E1 -29714.053,E2 -29714.053} C_VEL
LIN {X 0,Y 84.616,Z 445.855,A -85,B 0,C 180,E1 -29717.222,E2 -29717.222} C_VEL
LIN {X 0,Y 72.027,Z 452.395,A -85,B 0,C 180,E1 -29722.035,E2 -29722.035} C_VEL
LIN {X 0,Y 60.169,Z 457.495,A -85,B 0,C 180,E1 -29728.833,E2 -29728.833} C_VEL
LIN {X 0,Y 52.011,Z 460.429,A -85,B 0,C 180,E1 -29735.83,E2 -29735.83} C_VEL
LIN {X 0,Y 42.73,Z 463.288,A -85,B 0,C 180,E1 -29748.86,E2 -29748.86} C_VEL
LIN {X 0,Y 36.408,Z 464.993,A -85,B 0,C 180,E1 -29767.29,E2 -29767.29} C_VEL
LIN {X 0,Y 34.328,Z 465.579,A -85,B 0,C 180,E1 -29790.001,E2 -29790.001} C_VEL
LIN {X 0,Y 36.397,Z 465.021,A -85,B 0,C 180,E1 -29812.718,E2 -29812.718} C_VEL
LIN {X 0,Y 42.668,Z 463.353,A -85,B 0,C 180,E1 -29831.213,E2 -29831.213} C_VEL
LIN {X 0,Y 51.985,Z 460.525,A -85,B 0,C 180,E1 -29844.21,E2 -29844.21} C_VEL
LIN {X 0,Y 63.024,Z 456.468,A -85,B 0,C 180,E1 -29853.14,E2 -29853.14} C_VEL
LIN {X 0,Y 75.094,Z 451.081,A -85,B 0,C 180,E1 -29859.375,E2 -29859.375} C_VEL
LIN {X 0,Y 87.789,Z 444.208,A -85,B 0,C 180,E1 -29863.878,E2 -29863.878} C_VEL
LIN {X 0,Y 100.907,Z 435.62,A -85,B 0,C 180,E1 -29867.183,E2 -29867.183} C_VEL
LIN {X 0,Y 110.845,Z 427.909,A -85,B 0,C 180,E1 -29869.349,E2 -29869.349} C_VEL
LIN {X 0,Y 120.968,Z 418.809,A -85,B 0,C 180,E1 -29870.996,E2 -29870.996} C_VEL
LIN {X 0,Y 131.157,Z 408.075,A -85,B 0,C 180,E1 -29872.448,E2 -29872.448} C_VEL
LIN {X 0,Y 140.567,Z 396.348,A -85,B 0,C 180,E1 -29873.568,E2 -29873.568} C_VEL
LIN {X 0,Y 149.284,Z 383.293,A -85,B 0,C 180,E1 -29874.597,E2 -29874.597} C_VEL
LIN {X 0,Y 156.893,Z 369.389,A -85,B 0,C 180,E1 -29875.34,E2 -29875.34} C_VEL
LIN {X 0,Y 162.734,Z 356.116,A -85,B 0,C 180,E1 -29875.881,E2 -29875.881} C_VEL
LIN {X 0,Y 167.756,Z 341.418,A -85,B 0,C 180,E1 -29876.334,E2 -29876.334} C_VEL
LIN {X 0,Y 171.475,Z 326.332,A -85,B 0,C 180,E1 -29876.643,E2 -29876.643} C_VEL
LIN {X 0,Y 172.822,Z 318.694,A -85,B 0,C 180,E1 -29876.809,E2 -29876.809} C_VEL
LIN {X 0,Y 172.839,Z 316.983,A -85,B 0,C 180,E1 -29880,E2 -29880} C_VEL
LIN {X 0,Y 172.84,Z 318.687,A -85,B 0,C 180,E1 -29882.876,E2 -29882.876} C_VEL
LIN {X 0,Y 170.1,Z 332.835,A -85,B 0,C 180,E1 -29883.115,E2 -29883.115} C_VEL
LIN {X 0,Y 165.668,Z 348.376,A -85,B 0,C 180,E1 -29883.434,E2 -29883.434} C_VEL
LIN {X 0,Y 160.241,Z 362.515,A -85,B 0,C 180,E1 -29883.802,E2 -29883.802} C_VEL
LIN {X 0,Y 153.288,Z 376.744,A -85,B 0,C 180,E1 -29884.284,E2 -29884.284} C_VEL
LIN {X 0,Y 145.498,Z 389.716,A -85,B 0,C 180,E1 -29884.956,E2 -29884.956} C_VEL
LIN {X 0,Y 136.876,Z 401.71,A -85,B 0,C 180,E1 -29885.842,E2 -29885.842} C_VEL
LIN {X 0,Y 127.439,Z 412.816,A -85,B 0,C 180,E1 -29886.941,E2 -29886.941} C_VEL
LIN {X 0,Y 117.179,Z 423.048,A -85,B 0,C 180,E1 -29888.264,E2 -29888.264} C_VEL
LIN {X 0,Y 105.343,Z 433.052,A -85,B 0,C 180,E1 -29890.243,E2 -29890.243} C_VEL
LIN {X 0,Y 93.675,Z 441.368,A -85,B 0,C 180,E1 -29892.752,E2 -29892.752} C_VEL
LIN {X 0,Y 80.703,Z 449.193,A -85,B 0,C 180,E1 -29896.676,E2 -29896.676} C_VEL
LIN {X 0,Y 68.129,Z 455.418,A -85,B 0,C 180,E1 -29901.809,E2 -29901.809} C_VEL
LIN {X 0,Y 56.399,Z 460.245,A -85,B 0,C 180,E1 -29909.274,E2 -29909.274} C_VEL
LIN {X 0,Y 46.046,Z 463.792,A -85,B 0,C 180,E1 -29920.257,E2 -29920.257} C_VEL
LIN {X 0,Y 38.115,Z 466.135,A -85,B 0,C 180,E1 -29936.414,E2 -29936.414} C_VEL
LIN {X 0,Y 34.255,Z 467.33,A -85,B 0,C 180,E1 -29958.16,E2 -29958.16} C_VEL
LIN {X 0,Y 34.142,Z 467.496,A -85,B 0,C 180,E1 -29969.999,E2 -29969.999} C_VEL
LIN {X 0,Y 35.603,Z 466.851,A -85,B 0,C 180,E1 -29993.253,E2 -29993.253} C_VEL
LIN {X 0,Y 41.663,Z 465.054,A -85,B 0,C 180,E1 -30012.435,E2 -30012.435} C_VEL
LIN {X 0,Y 50.945,Z 462.088,A -85,B 0,C 180,E1 -30025.865,E2 -30025.865} C_VEL
LIN {X 0,Y 62.116,Z 457.888,A -85,B 0,C 180,E1 -30034.843,E2 -30034.843} C_VEL
LIN {X 0,Y 74.311,Z 452.342,A -85,B 0,C 180,E1 -30041.041,E2 -30041.041} C_VEL
LIN {X 0,Y 87.134,Z 445.302,A -85,B 0,C 180,E1 -30045.442,E2 -30045.442} C_VEL
LIN {X 0,Y 98.64,Z 437.779,A -85,B 0,C 180,E1 -30048.428,E2 -30048.428} C_VEL
LIN {X 0,Y 110.395,Z 428.722,A -85,B 0,C 180,E1 -30050.667,E2 -30050.667} C_VEL
LIN {X 0,Y 120.589,Z 419.48,A -85,B 0,C 180,E1 -30052.211,E2 -30052.211} C_VEL
LIN {X 0,Y 130.861,Z 408.597,A -85,B 0,C 180,E1 -30053.496,E2 -30053.496} C_VEL
LIN {X 0,Y 140.325,Z 396.706,A -85,B 0,C 180,E1 -30054.546,E2 -30054.546} C_VEL
LIN {X 0,Y 148.957,Z 383.721,A -85,B 0,C 180,E1 -30055.352,E2 -30055.352} C_VEL
LIN {X 0,Y 156.757,Z 369.357,A -85,B 0,C 180,E1 -30055.989,E2 -30055.989} C_VEL
LIN {X 0,Y 162.607,Z 355.93,A -85,B 0,C 180,E1 -30056.388,E2 -30056.388} C_VEL
LIN {X 0,Y 167.836,Z 340.297,A -85,B 0,C 180,E1 -30056.726,E2 -30056.726} C_VEL
LIN {X 0,Y 171.388,Z 325.25,A -85,B 0,C 180,E1 -30056.987,E2 -30056.987} C_VEL
LIN {X 0,Y 172.539,Z 318.454,A -85,B 0,C 180,E1 -30057.12,E2 -30057.12} C_VEL
LIN {X 0,Y 172.549,Z 316.623,A -85,B 0,C 180,E1 -30060,E2 -30060} C_VEL
LIN {X 0,Y 172.518,Z 318.373,A -85,B 0,C 180,E1 -30063.184,E2 -30063.184} C_VEL
LIN {X 0,Y 172.436,Z 319.295,A -85,B 0,C 180,E1 -30063.499,E2 -30063.499} C_VEL
LIN {X 0,Y 172.04,Z 321.769,A -85,B 0,C 180,E1 -30063.569,E2 -30063.569} C_VEL
LIN {X 0,Y 171.304,Z 325.33,A -85,B 0,C 180,E1 -30063.198,E2 -30063.198} C_VEL
LIN {X 0,Y 169.308,Z 333.686,A -85,B 0,C 180,E1 -30061.554,E2 -30061.554} C_VEL
LIN {X 0,Y 168.273,Z 337.588,A -85,B 0,C 180,E1 -30061.233,E2 -30061.233} C_VEL
LIN {X 0,Y 168.041,Z 338.385,A -85,B 0,C 180,E1 -30061.247,E2 -30061.247} C_VEL
LIN {X 0,Y 163.337,Z 352.96,A -85,B 0,C 180,E1 -30061.607,E2 -30061.607} C_VEL
LIN {X 0,Y 157.354,Z 367.113,A -85,B 0,C 180,E1 -30062.068,E2 -30062.068} C_VEL
LIN {X 0,Y 150.087,Z 380.811,A -85,B 0,C 180,E1 -30062.684,E2 -30062.684} C_VEL
LIN {X 0,Y 141.698,Z 393.745,A -85,B 0,C 180,E1 -30063.467,E2 -30063.467} C_VEL
LIN {X 0,Y 132.157,Z 405.94,A -85,B 0,C 180,E1 -30064.355,E2 -30064.355} C_VEL
LIN {X 0,Y 121.796,Z 417.05,A -85,B 0,C 180,E1 -30065.509,E2 -30065.509} C_VEL
LIN {X 0,Y 109.765,Z 427.834,A -85,B 0,C 180,E1 -30067.054,E2 -30067.054} C_VEL
LIN {X 0,Y 101.838,Z 433.927,A -85,B 0,C 180,E1 -30068.375,E2 -30068.375} C_VEL
LIN {X 0,Y 92.826,Z 440.108,A -85,B 0,C 180,E1 -30070.183,E2 -30070.183} C_VEL
LIN {X 0,Y 79.476,Z 447.851,A -85,B 0,C 180,E1 -30073.414,E2 -30073.414} C_VEL
LIN {X 0,Y 66.459,Z 454.006,A -85,B 0,C 180,E1 -30077.871,E2 -30077.871} C_VEL
LIN {X 0,Y 54.037,Z 458.746,A -85,B 0,C 180,E1 -30084.438,E2 -30084.438} C_VEL
LIN {X 0,Y 42.632,Z 462.209,A -85,B 0,C 180,E1 -30094.486,E2 -30094.486} C_VEL
LIN {X 0,Y 33.333,Z 464.481,A -85,B 0,C 180,E1 -30110.764,E2 -30110.764} C_VEL
LIN {X 0,Y 27.883,Z 465.627,A -85,B 0,C 180,E1 -30135.401,E2 -30135.401} C_VEL
LIN {X 0,Y 27.245,Z 465.777,A -85,B 0,C 180,E1 -30150.001,E2 -30150.001} C_VEL
LIN {X 0,Y 29.954,Z 465.22,A -85,B 0,C 180,E1 -30177.986,E2 -30177.986} C_VEL
LIN {X 0,Y 37.6,Z 463.553,A -85,B 0,C 180,E1 -30198.389,E2 -30198.389} C_VEL
LIN {X 0,Y 48.16,Z 460.724,A -85,B 0,C 180,E1 -30211.116,E2 -30211.116} C_VEL
LIN {X 0,Y 61.53,Z 456.116,A -85,B 0,C 180,E1 -30219.96,E2 -30219.96} C_VEL
LIN {X 0,Y 72.883,Z 451.28,A -85,B 0,C 180,E1 -30224.642,E2 -30224.642} C_VEL
LIN {X 0,Y 86.079,Z 444.407,A -85,B 0,C 180,E1 -30228.453,E2 -30228.453} C_VEL
LIN {X 0,Y 97.876,Z 437.014,A -85,B 0,C 180,E1 -30230.869,E2 -30230.869} C_VEL
LIN {X 0,Y 109.753,Z 428.106,A -85,B 0,C 180,E1 -30233.001,E2 -30233.001} C_VEL
LIN {X 0,Y 120.059,Z 419.006,A -85,B 0,C 180,E1 -30234.357,E2 -30234.357} C_VEL
LIN {X 0,Y 130.412,Z 408.271,A -85,B 0,C 180,E1 -30235.548,E2 -30235.548} C_VEL
LIN {X 0,Y 139.95,Z 396.543,A -85,B 0,C 180,E1 -30236.456,E2 -30236.456} C_VEL
LIN {X 0,Y 148.466,Z 384.006,A -85,B 0,C 180,E1 -30237.286,E2 -30237.286} C_VEL
LIN {X 0,Y 155.603,Z 371.344,A -85,B 0,C 180,E1 -30237.87,E2 -30237.87} C_VEL
LIN {X 0,Y 161.714,Z 358.024,A -85,B 0,C 180,E1 -30238.326,E2 -30238.326} C_VEL
LIN {X 0,Y 167.089,Z 342.871,A -85,B 0,C 180,E1 -30238.726,E2 -30238.726} C_VEL
LIN {X 0,Y 170.939,Z 327.906,A -85,B 0,C 180,E1 -30238.985,E2 -30238.985} C_VEL
LIN {X 0,Y 171.594,Z 324.489,A -85,B 0,C 180,E1 -30239.091,E2 -30239.091} C_VEL
LIN {X 0,Y 171.654,Z 324.137,A -85,B 0,C 180,E1 -30240,E2 -30240} C_VEL
LIN {X 0,Y 171.602,Z 324.501,A -85,B 0,C 180,E1 -30240.605,E2 -30240.605} C_VEL
LIN {X 0,Y 168.098,Z 339.452,A -85,B 0,C 180,E1 -30240.822,E2 -30240.822} C_VEL
LIN {X 0,Y 163.426,Z 353.727,A -85,B 0,C 180,E1 -30241.076,E2 -30241.076} C_VEL
LIN {X 0,Y 157.298,Z 368.073,A -85,B 0,C 180,E1 -30241.385,E2 -30241.385} C_VEL
LIN {X 0,Y 150.299,Z 381.207,A -85,B 0,C 180,E1 -30241.801,E2 -30241.801} C_VEL
LIN {X 0,Y 141.566,Z 394.599,A -85,B 0,C 180,E1 -30242.42,E2 -30242.42} C_VEL
LIN {X 0,Y 131.961,Z 406.833,A -85,B 0,C 180,E1 -30243.242,E2 -30243.242} C_VEL
LIN {X 0,Y 121.57,Z 417.955,A -85,B 0,C 180,E1 -30244.264,E2 -30244.264} C_VEL
LIN {X 0,Y 111.193,Z 427.345,A -85,B 0,C 180,E1 -30245.44,E2 -30245.44} C_VEL
LIN {X 0,Y 99.165,Z 436.583,A -85,B 0,C 180,E1 -30247.156,E2 -30247.156} C_VEL
LIN {X 0,Y 87.768,Z 443.99,A -85,B 0,C 180,E1 -30249.389,E2 -30249.389} C_VEL
LIN {X 0,Y 75.628,Z 450.666,A -85,B 0,C 180,E1 -30252.642,E2 -30252.642} C_VEL
LIN {X 0,Y 62.595,Z 456.541,A -85,B 0,C 180,E1 -30257.377,E2 -30257.377} C_VEL
LIN {X 0,Y 49.741,Z 461.227,A -85,B 0,C 180,E1 -30265.079,E2 -30265.079} C_VEL
LIN {X 0,Y 41.771,Z 463.592,A -85,B 0,C 180,E1 -30272.726,E2 -30272.726} C_VEL
LIN {X 0,Y 32.388,Z 465.935,A -85,B 0,C 180,E1 -30289.384,E2 -30289.384} C_VEL
LIN {X 0,Y 27.318,Z 467.13,A -85,B 0,C 180,E1 -30315.092,E2 -30315.092} C_VEL
LIN {X 0,Y 27.028,Z 467.297,A -85,B 0,C 180,E1 -30329.999,E2 -30329.999} C_VEL
LIN {X 0,Y 29.156,Z 466.651,A -85,B 0,C 180,E1 -30358.822,E2 -30358.822} C_VEL
LIN {X 0,Y 36.691,Z 464.852,A -85,B 0,C 180,E1 -30380.012,E2 -30380.012} C_VEL
LIN {X 0,Y 48.952,Z 461.366,A -85,B 0,C 180,E1 -30394.488,E2 -30394.488} C_VEL
LIN {X 0,Y 62.579,Z 456.429,A -85,B 0,C 180,E1 -30402.669,E2 -30402.669} C_VEL
LIN {X 0,Y 75.614,Z 450.513,A -85,B 0,C 180,E1 -30407.405,E2 -30407.405} C_VEL
LIN {X 0,Y 89.971,Z 442.464,A -85,B 0,C 180,E1 -30411.116,E2 -30411.116} C_VEL
LIN {X 0,Y 102.59,Z 433.873,A -85,B 0,C 180,E1 -30413.381,E2 -30413.381} C_VEL
LIN {X 0,Y 114.637,Z 424.079,A -85,B 0,C 180,E1 -30415.026,E2 -30415.026} C_VEL
LIN {X 0,Y 125.038,Z 414.071,A -85,B 0,C 180,E1 -30416.091,E2 -30416.091} C_VEL
LIN {X 0,Y 135.29,Z 402.398,A -85,B 0,C 180,E1 -30417.061,E2 -30417.061} C_VEL
LIN {X 0,Y 144.181,Z 390.327,A -85,B 0,C 180,E1 -30417.797,E2 -30417.797} C_VEL
LIN {X 0,Y 152.047,Z 377.523,A -85,B 0,C 180,E1 -30418.309,E2 -30418.309} C_VEL
LIN {X 0,Y 159.049,Z 363.541,A -85,B 0,C 180,E1 -30418.707,E2 -30418.707} C_VEL
LIN {X 0,Y 164.946,Z 348.52,A -85,B 0,C 180,E1 -30419.024,E2 -30419.024} C_VEL
LIN {X 0,Y 169.405,Z 333.153,A -85,B 0,C 180,E1 -30419.269,E2 -30419.269} C_VEL
LIN {X 0,Y 171.321,Z 324.19,A -85,B 0,C 180,E1 -30419.429,E2 -30419.429} C_VEL
LIN {X 0,Y 171.372,Z 323.828,A -85,B 0,C 180,E1 -30420,E2 -30420} C_VEL
LIN {X 0,Y 171.308,Z 324.198,A -85,B 0,C 180,E1 -30420.957,E2 -30420.957} C_VEL
LIN {X 0,Y 168.708,Z 335.982,A -85,B 0,C 180,E1 -30421.179,E2 -30421.179} C_VEL
LIN {X 0,Y 168.041,Z 338.385,A -85,B 0,C 180,E1 -30421.247,E2 -30421.247} C_VEL
LIN {X 0,Y 167.961,Z 338.961,A -85,B 0,C 180,E1 -30421.255,E2 -30421.255} C_VEL
LIN {X 0,Y 167.961,Z 406.978,A -85,B 0,C 180,E1 -30421.255,E2 -30421.255} C_VEL
LIN {X 0,Y 146.101,Z 406.978,A -85,B 0,C 180,E1 -30420.49,E2 -30420.49} C_VEL
LIN {X 0,Y 144.111,Z 404.978,A -85,B 0,C 180,E1 -30420.408,E2 -30420.408} C_VEL
LIN {X 0,Y 144.111,Z 396.328,A -85,B 0,C 180,E1 -30420.408,E2 -30420.408} C_VEL
LIN {X 0,Y 140.569,Z 395.117,A -85,B 0,C 180,E1 -30420.648,E2 -30420.648} C_VEL
LIN {X 0,Y 131.145,Z 406.877,A -85,B 0,C 180,E1 -30421.324,E2 -30421.324} C_VEL
LIN {X 0,Y 121.32,Z 417.251,A -85,B 0,C 180,E1 -30422.171,E2 -30422.171} C_VEL
LIN {X 0,Y 109.12,Z 428.035,A -85,B 0,C 180,E1 -30423.345,E2 -30423.345} C_VEL
LIN {X 0,Y 100.714,Z 434.363,A -85,B 0,C 180,E1 -30424.409,E2 -30424.409} C_VEL
LIN {X 0,Y 91.836,Z 440.309,A -85,B 0,C 180,E1 -30425.814,E2 -30425.814} C_VEL
LIN {X 0,Y 81.537,Z 446.257,A -85,B 0,C 180,E1 -30427.592,E2 -30427.592} C_VEL
LIN {X 0,Y 67.978,Z 452.796,A -85,B 0,C 180,E1 -30430.837,E2 -30430.837} C_VEL
LIN {X 0,Y 54.734,Z 457.896,A -85,B 0,C 180,E1 -30435.631,E2 -30435.631} C_VEL
LIN {X 0,Y 45.163,Z 460.83,A -85,B 0,C 180,E1 -30440.984,E2 -30440.984} C_VEL
LIN {X 0,Y 33.334,Z 463.688,A -85,B 0,C 180,E1 -30452.507,E2 -30452.507} C_VEL
LIN {X 0,Y 23.92,Z 465.392,A -85,B 0,C 180,E1 -30474.012,E2 -30474.012} C_VEL
LIN {X 0,Y 20.156,Z 465.975,A -85,B 0,C 180,E1 -30510.001,E2 -30510.001} C_VEL
LIN {X 0,Y 23.909,Z 465.419,A -85,B 0,C 180,E1 -30546.009,E2 -30546.009} C_VEL
LIN {X 0,Y 33.286,Z 463.752,A -85,B 0,C 180,E1 -30567.627,E2 -30567.627} C_VEL
LIN {X 0,Y 45.148,Z 460.923,A -85,B 0,C 180,E1 -30579.069,E2 -30579.069} C_VEL
LIN {X 0,Y 58.721,Z 456.591,A -85,B 0,C 180,E1 -30586.15,E2 -30586.15} C_VEL
LIN {X 0,Y 71.328,Z 451.478,A -85,B 0,C 180,E1 -30590.17,E2 -30590.17} C_VEL
LIN {X 0,Y 84.938,Z 444.605,A -85,B 0,C 180,E1 -30593.176,E2 -30593.176} C_VEL
LIN {X 0,Y 97,Z 437.212,A -85,B 0,C 180,E1 -30595.03,E2 -30595.03} C_VEL
LIN {X 0,Y 109.114,Z 428.303,A -85,B 0,C 180,E1 -30596.718,E2 -30596.718} C_VEL
